LIN {X 0,Y 397.144,Z 458.266,A -85,B 0,C 180,E1 -11410.353,E2 -11410.353} C_VEL
LIN {X 0,Y 397.162,Z 458.265,A -85,B 0,C 180,E1 -11413.553,E2 -11413.553} C_VEL
LIN {X 0,Y 397.225,Z 458.255,A -85,B 0,C 180,E1 -11416.703,E2 -11416.703} C_VEL
LIN {X 0,Y 397.225,Z 458.254,A -85,B 0,C 180,E1 -11419.809,E2 -11419.809} C_VEL
LIN {X 0,Y 397.361,Z 458.247,A -85,B 0,C 180,E1 -11422.888,E2 -11422.888} C_VEL
LIN {X 0,Y 397.221,Z 458.489,A -85,B 0,C 180,E1 -11425.433,E2 -11425.433} C_VEL
LIN {X 0,Y 397.512,Z 458.679,A -85,B 0,C 180,E1 -11427.974,E2 -11427.974} C_VEL
LIN {X 0,Y 397.666,Z 458.707,A -85,B 0,C 180,E1 -11430,E2 -11430} C_VEL
LIN {X 0,Y 397.415,Z 458.63,A -85,B 0,C 180,E1 -11433.041,E2 -11433.041} C_VEL
LIN {X 0,Y 397.361,Z 458.247,A -85,B 0,C 180,E1 -11437.112,E2 -11437.112} C_VEL
LIN {X 0,Y 397.225,Z 458.255,A -85,B 0,C 180,E1 -11440.191,E2 -11440.191} C_VEL
LIN {X 0,Y 397.223,Z 458.255,A -85,B 0,C 180,E1 -11443.321,E2 -11443.321} C_VEL
LIN {X 0,Y 397.178,Z 458.26,A -85,B 0,C 180,E1 -11447.155,E2 -11447.155} C_VEL
LIN {X 0,Y 397.098,Z 458.273,A -85,B 0,C 180,E1 -11450.73,E2 -11450.73} C_VEL
LIN {X 0,Y 397.128,Z 458.267,A -85,B 0,C 180,E1 -11454.018,E2 -11454.018} C_VEL
LIN {X 0,Y 397.129,Z 458.268,A -85,B 0,C 180,E1 -11456.332,E2 -11456.332} C_VEL
LIN {X 0,Y 396.46,Z 458.351,A -85,B 0,C 180,E1 -11457.179,E2 -11457.179} C_VEL
LIN {X 0,Y 393.585,Z 458.709,A -85,B 0,C 180,E1 -11458.555,E2 -11458.555} C_VEL
LIN {X 0,Y 391.146,Z 459.012,A -85,B 0,C 180,E1 -11459.666,E2 -11459.666} C_VEL
LIN {X 0,Y 390.094,Z 459.146,A -85,B 0,C 180,E1 -11460.526,E2 -11460.526} C_VEL
LIN {X 0,Y 390.006,Z 459.152,A -85,B 0,C 180,E1 -11460.817,E2 -11460.817} C_VEL
LIN {X 0,Y 390.062,Z 459.147,A -85,B 0,C 180,E1 -11464.024,E2 -11464.024} C_VEL
LIN {X 0,Y 390.041,Z 459.151,A -85,B 0,C 180,E1 -11467.551,E2 -11467.551} C_VEL
LIN {X 0,Y 390.07,Z 459.148,A -85,B 0,C 180,E1 -11470.825,E2 -11470.825} C_VEL
LIN {X 0,Y 390.053,Z 459.149,A -85,B 0,C 180,E1 -11473.887,E2 -11473.887} C_VEL
LIN {X 0,Y 390.111,Z 459.144,A -85,B 0,C 180,E1 -11476.798,E2 -11476.798} C_VEL
LIN {X 0,Y 390.071,Z 459.147,A -85,B 0,C 180,E1 -11479.563,E2 -11479.563} C_VEL
LIN {X 0,Y 390.053,Z 459.15,A -85,B 0,C 180,E1 -11482.446,E2 -11482.446} C_VEL
LIN {X 0,Y 390.06,Z 459.104,A -85,B 0,C 180,E1 -11486.045,E2 -11486.045} C_VEL
LIN {X 0,Y 390.044,Z 459.148,A -85,B 0,C 180,E1 -11489.867,E2 -11489.867} C_VEL
LIN {X 0,Y 390.105,Z 459.094,A -85,B 0,C 180,E1 -11493.232,E2 -11493.232} C_VEL
LIN {X 0,Y 390.068,Z 459.143,A -85,B 0,C 180,E1 -11496.761,E2 -11496.761} C_VEL
LIN {X 0,Y 390.095,Z 459.132,A -85,B 0,C 180,E1 -11499.983,E2 -11499.983} C_VEL
LIN {X 0,Y 390.129,Z 459.128,A -85,B 0,C 180,E1 -11503.248,E2 -11503.248} C_VEL
LIN {X 0,Y 390.186,Z 459.129,A -85,B 0,C 180,E1 -11506.562,E2 -11506.562} C_VEL
LIN {X 0,Y 390.197,Z 459.125,A -85,B 0,C 180,E1 -11510.671,E2 -11510.671} C_VEL
LIN {X 0,Y 390.32,Z 459.1,A -85,B 0,C 180,E1 -11513.798,E2 -11513.798} C_VEL
LIN {X 0,Y 390.412,Z 459.088,A -85,B 0,C 180,E1 -11517.937,E2 -11517.937} C_VEL
LIN {X 0,Y 390.541,Z 459.084,A -85,B 0,C 180,E1 -11520,E2 -11520} C_VEL
LIN {X 0,Y 390.308,Z 459.105,A -85,B 0,C 180,E1 -11523.097,E2 -11523.097} C_VEL
LIN {X 0,Y 390.327,Z 459.112,A -85,B 0,C 180,E1 -11526.202,E2 -11526.202} C_VEL
LIN {X 0,Y 390.197,Z 459.115,A -85,B 0,C 180,E1 -11529.329,E2 -11529.329} C_VEL
LIN {X 0,Y 390.163,Z 459.123,A -85,B 0,C 180,E1 -11532.483,E2 -11532.483} C_VEL
LIN {X 0,Y 390.131,Z 459.139,A -85,B 0,C 180,E1 -11535.677,E2 -11535.677} C_VEL
LIN {X 0,Y 390.097,Z 459.098,A -85,B 0,C 180,E1 -11538.923,E2 -11538.923} C_VEL
LIN {X 0,Y 390.029,Z 459.125,A -85,B 0,C 180,E1 -11542.235,E2 -11542.235} C_VEL
LIN {X 0,Y 390.112,Z 459.13,A -85,B 0,C 180,E1 -11545.744,E2 -11545.744} C_VEL
LIN {X 0,Y 390.058,Z 459.106,A -85,B 0,C 180,E1 -11549.11,E2 -11549.11} C_VEL
LIN {X 0,Y 390.049,Z 459.145,A -85,B 0,C 180,E1 -11552.721,E2 -11552.721} C_VEL
LIN {X 0,Y 390.051,Z 459.125,A -85,B 0,C 180,E1 -11555.826,E2 -11555.826} C_VEL
LIN {X 0,Y 390.069,Z 459.129,A -85,B 0,C 180,E1 -11559.22,E2 -11559.22} C_VEL
LIN {X 0,Y 390.115,Z 459.142,A -85,B 0,C 180,E1 -11562.387,E2 -11562.387} C_VEL
LIN {X 0,Y 390.057,Z 459.139,A -85,B 0,C 180,E1 -11565.358,E2 -11565.358} C_VEL
LIN {X 0,Y 390.056,Z 459.231,A -85,B 0,C 180,E1 -11567.74,E2 -11567.74} C_VEL
LIN {X 0,Y 390.768,Z 461.893,A -85,B 0,C 180,E1 -11568.518,E2 -11568.518} C_VEL
LIN {X 0,Y 393.681,Z 471.822,A -85,B 0,C 180,E1 -11571.078,E2 -11571.078} C_VEL
LIN {X 0,Y 395.714,Z 479.188,A -85,B 0,C 180,E1 -11572.82,E2 -11572.82} C_VEL
LIN {X 0,Y 403.295,Z 494.074,A -85,B 0,C 180,E1 -11573.969,E2 -11573.969} C_VEL
LIN {X 0,Y 409.389,Z 507.007,A -85,B 0,C 180,E1 -11574.853,E2 -11574.853} C_VEL
LIN {X 0,Y 414.14,Z 527.273,A -85,B 0,C 180,E1 -11575.728,E2 -11575.728} C_VEL
LIN {X 0,Y 410.722,Z 661.42,A -85,B 0,C 180,E1 -11578.145,E2 -11578.145} C_VEL
LIN {X 0,Y 409.788,Z 693.332,A -85,B 0,C 180,E1 -11578.749,E2 -11578.749} C_VEL
LIN {X 0,Y 408.893,Z 708.266,A -85,B 0,C 180,E1 -11579.158,E2 -11579.158} C_VEL
LIN {X 0,Y 407.444,Z 726.281,A -85,B 0,C 180,E1 -11579.862,E2 -11579.862} C_VEL
LIN {X 0,Y 405.925,Z 741.244,A -85,B 0,C 180,E1 -11580.648,E2 -11580.648} C_VEL
LIN {X 0,Y 404.496,Z 753.886,A -85,B 0,C 180,E1 -11581.459,E2 -11581.459} C_VEL
LIN {X 0,Y 402.955,Z 765.529,A -85,B 0,C 180,E1 -11582.331,E2 -11582.331} C_VEL
LIN {X 0,Y 401.258,Z 777.848,A -85,B 0,C 180,E1 -11583.418,E2 -11583.418} C_VEL
LIN {X 0,Y 399.674,Z 788.357,A -85,B 0,C 180,E1 -11584.481,E2 -11584.481} C_VEL
LIN {X 0,Y 398.093,Z 798.331,A -85,B 0,C 180,E1 -11585.628,E2 -11585.628} C_VEL
LIN {X 0,Y 396.444,Z 809.034,A -85,B 0,C 180,E1 -11587.046,E2 -11587.046} C_VEL
LIN {X 0,Y 394.852,Z 819.246,A -85,B 0,C 180,E1 -11588.6,E2 -11588.6} C_VEL
LIN {X 0,Y 393.427,Z 828.207,A -85,B 0,C 180,E1 -11590.16,E2 -11590.16} C_VEL
LIN {X 0,Y 392.277,Z 836.067,A -85,B 0,C 180,E1 -11591.721,E2 -11591.721} C_VEL
LIN {X 0,Y 391.408,Z 843.069,A -85,B 0,C 180,E1 -11593.305,E2 -11593.305} C_VEL
LIN {X 0,Y 390.552,Z 849.207,A -85,B 0,C 180,E1 -11594.875,E2 -11594.875} C_VEL
LIN {X 0,Y 389.788,Z 856.132,A -85,B 0,C 180,E1 -11596.968,E2 -11596.968} C_VEL
LIN {X 0,Y 389.223,Z 861.906,A -85,B 0,C 180,E1 -11599.071,E2 -11599.071} C_VEL
LIN {X 0,Y 388.948,Z 865.514,A -85,B 0,C 180,E1 -11600.641,E2 -11600.641} C_VEL
LIN {X 0,Y 388.809,Z 869.361,A -85,B 0,C 180,E1 -11602.731,E2 -11602.731} C_VEL
LIN {X 0,Y 388.736,Z 871.161,A -85,B 0,C 180,E1 -11603.905,E2 -11603.905} C_VEL
LIN {X 0,Y 388.656,Z 873.336,A -85,B 0,C 180,E1 -11605.852,E2 -11605.852} C_VEL
LIN {X 0,Y 388.649,Z 874.754,A -85,B 0,C 180,E1 -11607.927,E2 -11607.927} C_VEL
LIN {X 0,Y 388.671,Z 875.226,A -85,B 0,C 180,E1 -11610,E2 -11610} C_VEL
LIN {X 0,Y 388.649,Z 874.754,A -85,B 0,C 180,E1 -11612.073,E2 -11612.073} C_VEL
LIN {X 0,Y 388.656,Z 873.336,A -85,B 0,C 180,E1 -11614.148,E2 -11614.148} C_VEL
LIN {X 0,Y 388.757,Z 870.959,A -85,B 0,C 180,E1 -11616.227,E2 -11616.227} C_VEL
LIN {X 0,Y 388.897,Z 866.553,A -85,B 0,C 180,E1 -11618.836,E2 -11618.836} C_VEL
LIN {X 0,Y 389.063,Z 863.189,A -85,B 0,C 180,E1 -11620.407,E2 -11620.407} C_VEL
LIN {X 0,Y 389.627,Z 857.696,A -85,B 0,C 180,E1 -11622.501,E2 -11622.501} C_VEL
LIN {X 0,Y 390.134,Z 852.84,A -85,B 0,C 180,E1 -11624.075,E2 -11624.075} C_VEL
LIN {X 0,Y 391.062,Z 845.173,A -85,B 0,C 180,E1 -11626.174,E2 -11626.174} C_VEL
LIN {X 0,Y 391.964,Z 838.521,A -85,B 0,C 180,E1 -11627.746,E2 -11627.746} C_VEL
LIN {X 0,Y 393.005,Z 830.965,A -85,B 0,C 180,E1 -11629.319,E2 -11629.319} C_VEL
LIN {X 0,Y 394.321,Z 822.378,A -85,B 0,C 180,E1 -11630.883,E2 -11630.883} C_VEL
LIN {X 0,Y 395.742,Z 813.648,A -85,B 0,C 180,E1 -11632.282,E2 -11632.282} C_VEL
LIN {X 0,Y 397.465,Z 802.359,A -85,B 0,C 180,E1 -11633.858,E2 -11633.858} C_VEL
LIN {X 0,Y 398.918,Z 792.932,A -85,B 0,C 180,E1 -11635.012,E2 -11635.012} C_VEL
LIN {X 0,Y 400.659,Z 781.957,A -85,B 0,C 180,E1 -11636.184,E2 -11636.184} C_VEL
LIN {X 0,Y 402.337,Z 770.031,A -85,B 0,C 180,E1 -11637.292,E2 -11637.292} C_VEL
LIN {X 0,Y 403.98,Z 757.368,A -85,B 0,C 180,E1 -11638.298,E2 -11638.298} C_VEL
LIN {X 0,Y 405.41,Z 746.377,A -85,B 0,C 180,E1 -11639.038,E2 -11639.038} C_VEL
LIN {X 0,Y 406.742,Z 733.374,A -85,B 0,C 180,E1 -11639.785,E2 -11639.785} C_VEL
LIN {X 0,Y 408.03,Z 719.739,A -85,B 0,C 180,E1 -11640.414,E2 -11640.414} C_VEL
LIN {X 0,Y 409.047,Z 706.438,A -85,B 0,C 180,E1 -11640.895,E2 -11640.895} C_VEL
LIN {X 0,Y 409.807,Z 693.333,A -85,B 0,C 180,E1 -11641.249,E2 -11641.249} C_VEL
LIN {X 0,Y 410.809,Z 657.838,A -85,B 0,C 180,E1 -11641.919,E2 -11641.919} C_VEL
LIN {X 0,Y 414.182,Z 528.831,A -85,B 0,C 180,E1 -11644.236,E2 -11644.236} C_VEL
LIN {X 0,Y 413.765,Z 525.616,A -85,B 0,C 180,E1 -11644.341,E2 -11644.341} C_VEL
LIN {X 0,Y 409.15,Z 506.188,A -85,B 0,C 180,E1 -11645.187,E2 -11645.187} C_VEL
LIN {X 0,Y 399.516,Z 486.667,A -85,B 0,C 180,E1 -11646.585,E2 -11646.585} C_VEL
LIN {X 0,Y 395.6,Z 479.006,A -85,B 0,C 180,E1 -11647.209,E2 -11647.209} C_VEL
LIN {X 0,Y 392.819,Z 468.701,A -85,B 0,C 180,E1 -11649.707,E2 -11649.707} C_VEL
LIN {X 0,Y 390.089,Z 459.484,A -85,B 0,C 180,E1 -11652.144,E2 -11652.144} C_VEL
LIN {X 0,Y 390.037,Z 459.16,A -85,B 0,C 180,E1 -11652.373,E2 -11652.373} C_VEL
LIN {X 0,Y 390.097,Z 459.126,A -85,B 0,C 180,E1 -11656.106,E2 -11656.106} C_VEL
LIN {X 0,Y 390.077,Z 459.128,A -85,B 0,C 180,E1 -11659.174,E2 -11659.174} C_VEL
LIN {X 0,Y 390.041,Z 459.15,A -85,B 0,C 180,E1 -11662.448,E2 -11662.448} C_VEL
LIN {X 0,Y 390.062,Z 459.124,A -85,B 0,C 180,E1 -11666.045,E2 -11666.045} C_VEL
LIN {X 0,Y 390.041,Z 459.147,A -85,B 0,C 180,E1 -11668.497,E2 -11668.497} C_VEL
LIN {X 0,Y 390.111,Z 459.096,A -85,B 0,C 180,E1 -11672.069,E2 -11672.069} C_VEL
LIN {X 0,Y 390.07,Z 459.145,A -85,B 0,C 180,E1 -11675.519,E2 -11675.519} C_VEL
LIN {X 0,Y 390.047,Z 459.102,A -85,B 0,C 180,E1 -11678.877,E2 -11678.877} C_VEL
LIN {X 0,Y 390.12,Z 459.115,A -85,B 0,C 180,E1 -11682.166,E2 -11682.166} C_VEL
LIN {X 0,Y 390.136,Z 459.132,A -85,B 0,C 180,E1 -11685.392,E2 -11685.392} C_VEL
LIN {X 0,Y 390.142,Z 459.138,A -85,B 0,C 180,E1 -11688.571,E2 -11688.571} C_VEL
LIN {X 0,Y 390.3,Z 459.103,A -85,B 0,C 180,E1 -11692.031,E2 -11692.031} C_VEL
LIN {X 0,Y 390.223,Z 459.122,A -85,B 0,C 180,E1 -11694.833,E2 -11694.833} C_VEL
LIN {X 0,Y 390.412,Z 459.097,A -85,B 0,C 180,E1 -11697.937,E2 -11697.937} C_VEL
LIN {X 0,Y 390.541,Z 459.083,A -85,B 0,C 180,E1 -11700,E2 -11700} C_VEL
LIN {X 0,Y 390.308,Z 459.113,A -85,B 0,C 180,E1 -11703.096,E2 -11703.096} C_VEL
LIN {X 0,Y 390.295,Z 459.102,A -85,B 0,C 180,E1 -11706.61,E2 -11706.61} C_VEL
LIN {X 0,Y 390.197,Z 459.124,A -85,B 0,C 180,E1 -11709.329,E2 -11709.329} C_VEL
LIN {X 0,Y 390.186,Z 459.129,A -85,B 0,C 180,E1 -11713.438,E2 -11713.438} C_VEL
LIN {X 0,Y 390.14,Z 459.137,A -85,B 0,C 180,E1 -11717.308,E2 -11717.308} C_VEL
LIN {X 0,Y 390.079,Z 459.133,A -85,B 0,C 180,E1 -11720.47,E2 -11720.47} C_VEL
LIN {X 0,Y 390.065,Z 459.142,A -85,B 0,C 180,E1 -11723.352,E2 -11723.352} C_VEL
LIN {X 0,Y 390.105,Z 459.094,A -85,B 0,C 180,E1 -11726.768,E2 -11726.768} C_VEL
LIN {X 0,Y 390.036,Z 459.15,A -85,B 0,C 180,E1 -11730.299,E2 -11730.299} C_VEL
LIN {X 0,Y 390.06,Z 459.104,A -85,B 0,C 180,E1 -11734.025,E2 -11734.025} C_VEL
LIN {X 0,Y 390.053,Z 459.15,A -85,B 0,C 180,E1 -11737.554,E2 -11737.554} C_VEL
LIN {X 0,Y 390.076,Z 459.147,A -85,B 0,C 180,E1 -11740.826,E2 -11740.826} C_VEL
LIN {X 0,Y 390.099,Z 459.143,A -85,B 0,C 180,E1 -11743.894,E2 -11743.894} C_VEL
LIN {X 0,Y 390.074,Z 459.148,A -85,B 0,C 180,E1 -11747.62,E2 -11747.62} C_VEL
LIN {X 0,Y 390.089,Z 459.146,A -85,B 0,C 180,E1 -11750.909,E2 -11750.909} C_VEL
LIN {X 0,Y 390.08,Z 459.145,A -85,B 0,C 180,E1 -11754.794,E2 -11754.794} C_VEL
LIN {X 0,Y 390.018,Z 459.152,A -85,B 0,C 180,E1 -11758.496,E2 -11758.496} C_VEL
LIN {X 0,Y 390.112,Z 459.143,A -85,B 0,C 180,E1 -11762.07,E2 -11762.07} C_VEL
LIN {X 0,Y 390.076,Z 459.145,A -85,B 0,C 180,E1 -11765.52,E2 -11765.52} C_VEL
LIN {X 0,Y 390.051,Z 459.149,A -85,B 0,C 180,E1 -11768.878,E2 -11768.878} C_VEL
LIN {X 0,Y 390.124,Z 459.142,A -85,B 0,C 180,E1 -11772.167,E2 -11772.167} C_VEL
LIN {X 0,Y 390.173,Z 459.305,A -85,B 0,C 180,E1 -11775.527,E2 -11775.527} C_VEL
LIN {X 0,Y 390.554,Z 460.669,A -85,B 0,C 180,E1 -11776.957,E2 -11776.957} C_VEL
LIN {X 0,Y 391.562,Z 462.574,A -85,B 0,C 180,E1 -11778.351,E2 -11778.351} C_VEL
LIN {X 0,Y 392.987,Z 463.95,A -85,B 0,C 180,E1 -11780.31,E2 -11780.31} C_VEL
LIN {X 0,Y 394.469,Z 464.73,A -85,B 0,C 180,E1 -11782.836,E2 -11782.836} C_VEL
LIN {X 0,Y 395.521,Z 465.381,A -85,B 0,C 180,E1 -11785.414,E2 -11785.414} C_VEL
LIN {X 0,Y 396.123,Z 465.642,A -85,B 0,C 180,E1 -11787.967,E2 -11787.967} C_VEL
LIN {X 0,Y 396.315,Z 465.672,A -85,B 0,C 180,E1 -11790,E2 -11790} C_VEL
LIN {X 0,Y 396.123,Z 465.642,A -85,B 0,C 180,E1 -11792.033,E2 -11792.033} C_VEL
LIN {X 0,Y 395.52,Z 465.38,A -85,B 0,C 180,E1 -11794.586,E2 -11794.586} C_VEL
LIN {X 0,Y 394.468,Z 464.729,A -85,B 0,C 180,E1 -11797.164,E2 -11797.164} C_VEL
LIN {X 0,Y 392.881,Z 463.843,A -85,B 0,C 180,E1 -11799.836,E2 -11799.836} C_VEL
LIN {X 0,Y 391.466,Z 462.435,A -85,B 0,C 180,E1 -11801.783,E2 -11801.783} C_VEL
LIN {X 0,Y 390.268,Z 459.788,A -85,B 0,C 180,E1 -11803.804,E2 -11803.804} C_VEL
LIN {X 0,Y 390.125,Z 459.18,A -85,B 0,C 180,E1 -11805.142,E2 -11805.142} C_VEL
LIN {X 0,Y 390.124,Z 459.141,A -85,B 0,C 180,E1 -11807.833,E2 -11807.833} C_VEL
LIN {X 0,Y 390.051,Z 459.149,A -85,B 0,C 180,E1 -11811.122,E2 -11811.122} C_VEL
LIN {X 0,Y 390.075,Z 459.146,A -85,B 0,C 180,E1 -11814.48,E2 -11814.48} C_VEL
LIN {X 0,Y 390.112,Z 459.143,A -85,B 0,C 180,E1 -11817.93,E2 -11817.93} C_VEL
LIN {X 0,Y 390.006,Z 459.152,A -85,B 0,C 180,E1 -11820.817,E2 -11820.817} C_VEL
LIN {X 0,Y 389.333,Z 459.239,A -85,B 0,C 180,E1 -11821.679,E2 -11821.679} C_VEL
LIN {X 0,Y 386.485,Z 459.594,A -85,B 0,C 180,E1 -11823.081,E2 -11823.081} C_VEL
LIN {X 0,Y 384.087,Z 459.891,A -85,B 0,C 180,E1 -11824.214,E2 -11824.214} C_VEL
LIN {X 0,Y 383.07,Z 460.019,A -85,B 0,C 180,E1 -11825.09,E2 -11825.09} C_VEL
LIN {X 0,Y 382.993,Z 460.025,A -85,B 0,C 180,E1 -11825.386,E2 -11825.386} C_VEL
LIN {X 0,Y 383.002,Z 460.027,A -85,B 0,C 180,E1 -11828.6,E2 -11828.6} C_VEL
LIN {X 0,Y 383.007,Z 460.025,A -85,B 0,C 180,E1 -11831.343,E2 -11831.343} C_VEL
LIN {X 0,Y 383.001,Z 460.027,A -85,B 0,C 180,E1 -11834.305,E2 -11834.305} C_VEL
LIN {X 0,Y 383.068,Z 460.02,A -85,B 0,C 180,E1 -11837.249,E2 -11837.249} C_VEL
LIN {X 0,Y 383.015,Z 460.026,A -85,B 0,C 180,E1 -11840.412,E2 -11840.412} C_VEL
LIN {X 0,Y 383.019,Z 460.006,A -85,B 0,C 180,E1 -11844.044,E2 -11844.044} C_VEL
LIN {X 0,Y 382.98,Z 460.004,A -85,B 0,C 180,E1 -11847.577,E2 -11847.577} C_VEL
LIN {X 0,Y 382.99,Z 460.027,A -85,B 0,C 180,E1 -11850.3,E2 -11850.3} C_VEL
LIN {X 0,Y 383.049,Z 459.974,A -85,B 0,C 180,E1 -11852.698,E2 -11852.698} C_VEL
LIN {X 0,Y 383.042,Z 459.992,A -85,B 0,C 180,E1 -11855.039,E2 -11855.039} C_VEL
LIN {X 0,Y 382.984,Z 460.026,A -85,B 0,C 180,E1 -11858.469,E2 -11858.469} C_VEL
LIN {X 0,Y 383.081,Z 460.016,A -85,B 0,C 180,E1 -11861.828,E2 -11861.828} C_VEL
LIN {X 0,Y 383.101,Z 460.003,A -85,B 0,C 180,E1 -11865.118,E2 -11865.118} C_VEL
LIN {X 0,Y 383.089,Z 460.001,A -85,B 0,C 180,E1 -11868.358,E2 -11868.358} C_VEL
LIN {X 0,Y 383.256,Z 459.988,A -85,B 0,C 180,E1 -11871.975,E2 -11871.975} C_VEL
LIN {X 0,Y 383.193,Z 459.993,A -85,B 0,C 180,E1 -11874.739,E2 -11874.739} C_VEL
LIN {X 0,Y 383.38,Z 459.964,A -85,B 0,C 180,E1 -11877.899,E2 -11877.899} C_VEL
LIN {X 0,Y 383.511,Z 459.96,A -85,B 0,C 180,E1 -11880,E2 -11880} C_VEL
LIN {X 0,Y 383.244,Z 459.984,A -85,B 0,C 180,E1 -11883.154,E2 -11883.154} C_VEL
LIN {X 0,Y 383.281,Z 459.989,A -85,B 0,C 180,E1 -11886.317,E2 -11886.317} C_VEL
LIN {X 0,Y 383.144,Z 459.996,A -85,B 0,C 180,E1 -11889.502,E2 -11889.502} C_VEL
LIN {X 0,Y 383.118,Z 459.997,A -85,B 0,C 180,E1 -11893.536,E2 -11893.536} C_VEL
LIN {X 0,Y 383.087,Z 459.997,A -85,B 0,C 180,E1 -11897.455,E2 -11897.455} C_VEL
LIN {X 0,Y 383.021,Z 459.97,A -85,B 0,C 180,E1 -11900.647,E2 -11900.647} C_VEL
LIN {X 0,Y 383.018,Z 460.023,A -85,B 0,C 180,E1 -11903.808,E2 -11903.808} C_VEL
LIN {X 0,Y 383.073,Z 460,A -85,B 0,C 180,E1 -11906.124,E2 -11906.124} C_VEL
LIN {X 0,Y 383.043,Z 459.974,A -85,B 0,C 180,E1 -11908.493,E2 -11908.493} C_VEL
LIN {X 0,Y 383.002,Z 460.025,A -85,B 0,C 180,E1 -11912.428,E2 -11912.428} C_VEL
LIN {X 0,Y 383.021,Z 460.001,A -85,B 0,C 180,E1 -11915.956,E2 -11915.956} C_VEL
LIN {X 0,Y 383.017,Z 460.003,A -85,B 0,C 180,E1 -11919.588,E2 -11919.588} C_VEL
LIN {X 0,Y 383.061,Z 460.016,A -85,B 0,C 180,E1 -11922.789,E2 -11922.789} C_VEL
LIN {X 0,Y 383.01,Z 460.02,A -85,B 0,C 180,E1 -11926.522,E2 -11926.522} C_VEL
LIN {X 0,Y 383.036,Z 460.276,A -85,B 0,C 180,E1 -11927.147,E2 -11927.147} C_VEL
LIN {X 0,Y 386.351,Z 471.502,A -85,B 0,C 180,E1 -11930.189,E2 -11930.189} C_VEL
LIN {X 0,Y 388.322,Z 478.732,A -85,B 0,C 180,E1 -11931.974,E2 -11931.974} C_VEL
LIN {X 0,Y 397.62,Z 496.664,A -85,B 0,C 180,E1 -11933.433,E2 -11933.433} C_VEL
LIN {X 0,Y 403.932,Z 510.042,A -85,B 0,C 180,E1 -11934.376,E2 -11934.376} C_VEL
LIN {X 0,Y 408.265,Z 528.969,A -85,B 0,C 180,E1 -11935.204,E2 -11935.204} C_VEL
LIN {X 0,Y 404.323,Z 675.539,A -85,B 0,C 180,E1 -11937.875,E2 -11937.875} C_VEL
LIN {X 0,Y 403.49,Z 698.576,A -85,B 0,C 180,E1 -11938.352,E2 -11938.352} C_VEL
LIN {X 0,Y 402.19,Z 715.47,A -85,B 0,C 180,E1 -11938.903,E2 -11938.903} C_VEL
LIN {X 0,Y 401.069,Z 728.224,A -85,B 0,C 180,E1 -11939.459,E2 -11939.459} C_VEL
LIN {X 0,Y 399.722,Z 741.033,A -85,B 0,C 180,E1 -11940.146,E2 -11940.146} C_VEL
LIN {X 0,Y 398.23,Z 753.675,A -85,B 0,C 180,E1 -11940.967,E2 -11940.967} C_VEL
LIN {X 0,Y 396.63,Z 765.317,A -85,B 0,C 180,E1 -11941.851,E2 -11941.851} C_VEL
LIN {X 0,Y 394.824,Z 777.635,A -85,B 0,C 180,E1 -11942.95,E2 -11942.95} C_VEL
LIN {X 0,Y 393.218,Z 788.145,A -85,B 0,C 180,E1 -11944.031,E2 -11944.031} C_VEL
LIN {X 0,Y 391.37,Z 799.125,A -85,B 0,C 180,E1 -11945.323,E2 -11945.323} C_VEL
LIN {X 0,Y 389.803,Z 808.82,A -85,B 0,C 180,E1 -11946.632,E2 -11946.632} C_VEL
LIN {X 0,Y 388.132,Z 819.033,A -85,B 0,C 180,E1 -11948.211,E2 -11948.211} C_VEL
LIN {X 0,Y 386.63,Z 827.993,A -85,B 0,C 180,E1 -11949.796,E2 -11949.796} C_VEL
LIN {X 0,Y 385.34,Z 836.439,A -85,B 0,C 180,E1 -11951.513,E2 -11951.513} C_VEL
LIN {X 0,Y 384.323,Z 843.908,A -85,B 0,C 180,E1 -11953.261,E2 -11953.261} C_VEL
LIN {X 0,Y 383.353,Z 850.811,A -85,B 0,C 180,E1 -11955.128,E2 -11955.128} C_VEL
LIN {X 0,Y 382.823,Z 855.709,A -85,B 0,C 180,E1 -11956.653,E2 -11956.653} C_VEL
LIN {X 0,Y 382.318,Z 860.408,A -85,B 0,C 180,E1 -11958.334,E2 -11958.334} C_VEL
LIN {X 0,Y 381.887,Z 865.303,A -85,B 0,C 180,E1 -11960.466,E2 -11960.466} C_VEL
LIN {X 0,Y 381.711,Z 869.149,A -85,B 0,C 180,E1 -11962.595,E2 -11962.595} C_VEL
LIN {X 0,Y 381.655,Z 871.134,A -85,B 0,C 180,E1 -11963.924,E2 -11963.924} C_VEL
LIN {X 0,Y 381.581,Z 873.126,A -85,B 0,C 180,E1 -11965.775,E2 -11965.775} C_VEL
LIN {X 0,Y 381.547,Z 874.544,A -85,B 0,C 180,E1 -11967.889,E2 -11967.889} C_VEL
LIN {X 0,Y 381.586,Z 875.016,A -85,B 0,C 180,E1 -11970,E2 -11970} C_VEL
LIN {X 0,Y 381.547,Z 874.544,A -85,B 0,C 180,E1 -11972.111,E2 -11972.111} C_VEL
LIN {X 0,Y 381.581,Z 873.126,A -85,B 0,C 180,E1 -11974.225,E2 -11974.225} C_VEL
LIN {X 0,Y 381.662,Z 870.748,A -85,B 0,C 180,E1 -11976.343,E2 -11976.343} C_VEL
LIN {X 0,Y 381.819,Z 866.341,A -85,B 0,C 180,E1 -11979.001,E2 -11979.001} C_VEL
LIN {X 0,Y 382.021,Z 862.977,A -85,B 0,C 180,E1 -11980.601,E2 -11980.601} C_VEL
LIN {X 0,Y 382.59,Z 857.483,A -85,B 0,C 180,E1 -11982.734,E2 -11982.734} C_VEL
LIN {X 0,Y 383.157,Z 852.627,A -85,B 0,C 180,E1 -11984.336,E2 -11984.336} C_VEL
LIN {X 0,Y 384.151,Z 844.96,A -85,B 0,C 180,E1 -11986.473,E2 -11986.473} C_VEL
LIN {X 0,Y 385.082,Z 838.307,A -85,B 0,C 180,E1 -11988.075,E2 -11988.075} C_VEL
LIN {X 0,Y 386.184,Z 830.751,A -85,B 0,C 180,E1 -11989.674,E2 -11989.674} C_VEL
LIN {X 0,Y 387.58,Z 822.165,A -85,B 0,C 180,E1 -11991.263,E2 -11991.263} C_VEL
LIN {X 0,Y 389.242,Z 812.49,A -85,B 0,C 180,E1 -11992.823,E2 -11992.823} C_VEL
LIN {X 0,Y 390.871,Z 802.146,A -85,B 0,C 180,E1 -11994.286,E2 -11994.286} C_VEL
LIN {X 0,Y 392.409,Z 792.72,A -85,B 0,C 180,E1 -11995.457,E2 -11995.457} C_VEL
LIN {X 0,Y 394.393,Z 780.55,A -85,B 0,C 180,E1 -11996.763,E2 -11996.763} C_VEL
LIN {X 0,Y 396.139,Z 768.316,A -85,B 0,C 180,E1 -11997.899,E2 -11997.899} C_VEL
LIN {X 0,Y 397.693,Z 757.156,A -85,B 0,C 180,E1 -11998.787,E2 -11998.787} C_VEL
LIN {X 0,Y 399.277,Z 745.139,A -85,B 0,C 180,E1 -11999.6,E2 -11999.6} C_VEL
LIN {X 0,Y 400.569,Z 733.163,A -85,B 0,C 180,E1 -12000.292,E2 -12000.292} C_VEL
LIN {X 0,Y 401.864,Z 719.795,A -85,B 0,C 180,E1 -12000.919,E2 -12000.919} C_VEL
LIN {X 0,Y 402.944,Z 706.567,A -85,B 0,C 180,E1 -12001.403,E2 -12001.403} C_VEL
LIN {X 0,Y 403.749,Z 693.123,A -85,B 0,C 180,E1 -12001.772,E2 -12001.772} C_VEL
LIN {X 0,Y 404.797,Z 657.628,A -85,B 0,C 180,E1 -12002.451,E2 -12002.451} C_VEL
LIN {X 0,Y 408.007,Z 538.652,A -85,B 0,C 180,E1 -12004.618,E2 -12004.618} C_VEL
LIN {X 0,Y 408.138,Z 528.273,A -85,B 0,C 180,E1 -12004.823,E2 -12004.823} C_VEL
LIN {X 0,Y 403.786,Z 509.589,A -85,B 0,C 180,E1 -12005.649,E2 -12005.649} C_VEL
LIN {X 0,Y 394.84,Z 491.255,A -85,B 0,C 180,E1 -12006.985,E2 -12006.985} C_VEL
LIN {X 0,Y 388.337,Z 478.732,A -85,B 0,C 180,E1 -12008.024,E2 -12008.024} C_VEL
LIN {X 0,Y 385.267,Z 467.825,A -85,B 0,C 180,E1 -12010.778,E2 -12010.778} C_VEL
LIN {X 0,Y 383.061,Z 460.454,A -85,B 0,C 180,E1 -12012.788,E2 -12012.788} C_VEL
LIN {X 0,Y 383.027,Z 460.016,A -85,B 0,C 180,E1 -12013.114,E2 -12013.114} C_VEL
LIN {X 0,Y 383.033,Z 460.004,A -85,B 0,C 180,E1 -12015.794,E2 -12015.794} C_VEL
LIN {X 0,Y 383.039,Z 460.009,A -85,B 0,C 180,E1 -12018.786,E2 -12018.786} C_VEL
LIN {X 0,Y 382.998,Z 460.028,A -85,B 0,C 180,E1 -12022.095,E2 -12022.095} C_VEL
LIN {X 0,Y 383.012,Z 459.995,A -85,B 0,C 180,E1 -12025.331,E2 -12025.331} C_VEL
LIN {X 0,Y 383.03,Z 460.025,A -85,B 0,C 180,E1 -12027.852,E2 -12027.852} C_VEL
LIN {X 0,Y 383.057,Z 459.972,A -85,B 0,C 180,E1 -12031.72,E2 -12031.72} C_VEL
LIN {X 0,Y 383.044,Z 460.019,A -85,B 0,C 180,E1 -12035.039,E2 -12035.039} C_VEL
LIN {X 0,Y 382.984,Z 459.987,A -85,B 0,C 180,E1 -12038.468,E2 -12038.468} C_VEL
LIN {X 0,Y 383.081,Z 459.986,A -85,B 0,C 180,E1 -12041.827,E2 -12041.827} C_VEL
LIN {X 0,Y 383.102,Z 460.008,A -85,B 0,C 180,E1 -12045.118,E2 -12045.118} C_VEL
LIN {X 0,Y 383.091,Z 460.012,A -85,B 0,C 180,E1 -12048.358,E2 -12048.358} C_VEL
LIN {X 0,Y 383.256,Z 459.979,A -85,B 0,C 180,E1 -12051.975,E2 -12051.975} C_VEL
LIN {X 0,Y 383.195,Z 459.998,A -85,B 0,C 180,E1 -12054.738,E2 -12054.738} C_VEL
LIN {X 0,Y 383.379,Z 459.973,A -85,B 0,C 180,E1 -12057.899,E2 -12057.899} C_VEL
LIN {X 0,Y 383.511,Z 459.958,A -85,B 0,C 180,E1 -12060,E2 -12060} C_VEL
LIN {X 0,Y 383.245,Z 459.992,A -85,B 0,C 180,E1 -12063.153,E2 -12063.153} C_VEL
LIN {X 0,Y 383.255,Z 459.978,A -85,B 0,C 180,E1 -12066.602,E2 -12066.602} C_VEL
LIN {X 0,Y 383.143,Z 460.002,A -85,B 0,C 180,E1 -12069.502,E2 -12069.502} C_VEL
LIN {X 0,Y 383.117,Z 460.009,A -85,B 0,C 180,E1 -12073.536,E2 -12073.536} C_VEL
LIN {X 0,Y 383.086,Z 460.015,A -85,B 0,C 180,E1 -12077.454,E2 -12077.454} C_VEL
LIN {X 0,Y 383.02,Z 460.012,A -85,B 0,C 180,E1 -12080.647,E2 -12080.647} C_VEL
LIN {X 0,Y 383.017,Z 460.018,A -85,B 0,C 180,E1 -12083.808,E2 -12083.808} C_VEL
LIN {X 0,Y 383.072,Z 459.97,A -85,B 0,C 180,E1 -12086.123,E2 -12086.123} C_VEL
LIN {X 0,Y 383.042,Z 459.996,A -85,B 0,C 180,E1 -12088.492,E2 -12088.492} C_VEL
LIN {X 0,Y 383.003,Z 460.008,A -85,B 0,C 180,E1 -12092.15,E2 -12092.15} C_VEL
LIN {X 0,Y 383.01,Z 459.984,A -85,B 0,C 180,E1 -12094.668,E2 -12094.668} C_VEL
LIN {X 0,Y 383.003,Z 460.027,A -85,B 0,C 180,E1 -12097.906,E2 -12097.906} C_VEL
LIN {X 0,Y 383.04,Z 460.024,A -85,B 0,C 180,E1 -12101.339,E2 -12101.339} C_VEL
LIN {X 0,Y 383.03,Z 460.023,A -85,B 0,C 180,E1 -12104.31,E2 -12104.31} C_VEL
LIN {X 0,Y 383.033,Z 460.023,A -85,B 0,C 180,E1 -12107.245,E2 -12107.245} C_VEL
LIN {X 0,Y 383.015,Z 460.025,A -85,B 0,C 180,E1 -12110.413,E2 -12110.413} C_VEL
LIN {X 0,Y 383.021,Z 460.024,A -85,B 0,C 180,E1 -12114.045,E2 -12114.045} C_VEL
LIN {X 0,Y 382.981,Z 460.03,A -85,B 0,C 180,E1 -12117.578,E2 -12117.578} C_VEL
LIN {X 0,Y 382.987,Z 460.028,A -85,B 0,C 180,E1 -12120.3,E2 -12120.3} C_VEL
LIN {X 0,Y 383.076,Z 460.017,A -85,B 0,C 180,E1 -12124.021,E2 -12124.021} C_VEL
LIN {X 0,Y 383.004,Z 460.026,A -85,B 0,C 180,E1 -12127.336,E2 -12127.336} C_VEL
LIN {X 0,Y 383.089,Z 460.2,A -85,B 0,C 180,E1 -12130.021,E2 -12130.021} C_VEL
LIN {X 0,Y 383.447,Z 461.553,A -85,B 0,C 180,E1 -12131.015,E2 -12131.015} C_VEL
LIN {X 0,Y 384.784,Z 463.815,A -85,B 0,C 180,E1 -12132.232,E2 -12132.232} C_VEL
LIN {X 0,Y 386.964,Z 465.493,A -85,B 0,C 180,E1 -12134.192,E2 -12134.192} C_VEL
LIN {X 0,Y 388.846,Z 466.639,A -85,B 0,C 180,E1 -12136.011,E2 -12136.011} C_VEL
LIN {X 0,Y 390.564,Z 469.516,A -85,B 0,C 180,E1 -12138.189,E2 -12138.189} C_VEL
LIN {X 0,Y 392.123,Z 470.995,A -85,B 0,C 180,E1 -12140.317,E2 -12140.317} C_VEL
LIN {X 0,Y 393.591,Z 471.775,A -85,B 0,C 180,E1 -12142.82,E2 -12142.82} C_VEL
LIN {X 0,Y 394.492,Z 472.245,A -85,B 0,C 180,E1 -12144.89,E2 -12144.89} C_VEL
LIN {X 0,Y 394.837,Z 472.584,A -85,B 0,C 180,E1 -12145.917,E2 -12145.917} C_VEL
LIN {X 0,Y 395.257,Z 472.689,A -85,B 0,C 180,E1 -12147.962,E2 -12147.962} C_VEL
LIN {X 0,Y 395.45,Z 472.72,A -85,B 0,C 180,E1 -12150,E2 -12150} C_VEL
LIN {X 0,Y 395.258,Z 472.69,A -85,B 0,C 180,E1 -12152.038,E2 -12152.038} C_VEL
LIN {X 0,Y 394.65,Z 472.428,A -85,B 0,C 180,E1 -12154.596,E2 -12154.596} C_VEL
LIN {X 0,Y 393.591,Z 471.772,A -85,B 0,C 180,E1 -12157.18,E2 -12157.18} C_VEL
LIN {X 0,Y 391.99,Z 470.903,A -85,B 0,C 180,E1 -12159.859,E2 -12159.859} C_VEL
LIN {X 0,Y 390.47,Z 469.378,A -85,B 0,C 180,E1 -12161.946,E2 -12161.946} C_VEL
LIN {X 0,Y 388.845,Z 466.637,A -85,B 0,C 180,E1 -12163.989,E2 -12163.989} C_VEL
LIN {X 0,Y 386.032,Z 464.937,A -85,B 0,C 180,E1 -12166.662,E2 -12166.662} C_VEL
LIN {X 0,Y 384.202,Z 463.095,A -85,B 0,C 180,E1 -12168.255,E2 -12168.255} C_VEL
LIN {X 0,Y 383.196,Z 460.804,A -85,B 0,C 180,E1 -12169.415,E2 -12169.415} C_VEL
LIN {X 0,Y 383.051,Z 460.065,A -85,B 0,C 180,E1 -12170.401,E2 -12170.401} C_VEL
LIN {X 0,Y 383.029,Z 460.024,A -85,B 0,C 180,E1 -12173.807,E2 -12173.807} C_VEL
LIN {X 0,Y 383.075,Z 460.019,A -85,B 0,C 180,E1 -12176.123,E2 -12176.123} C_VEL
LIN {X 0,Y 382.987,Z 460.028,A -85,B 0,C 180,E1 -12179.7,E2 -12179.7} C_VEL
LIN {X 0,Y 382.998,Z 460.029,A -85,B 0,C 180,E1 -12183.4,E2 -12183.4} C_VEL
LIN {X 0,Y 382.993,Z 460.025,A -85,B 0,C 180,E1 -12185.386,E2 -12185.386} C_VEL
LIN {X 0,Y 382.353,Z 460.109,A -85,B 0,C 180,E1 -12186.264,E2 -12186.264} C_VEL
LIN {X 0,Y 379.545,Z 460.459,A -85,B 0,C 180,E1 -12187.692,E2 -12187.692} C_VEL
LIN {X 0,Y 377.14,Z 460.758,A -85,B 0,C 180,E1 -12188.846,E2 -12188.846} C_VEL
LIN {X 0,Y 376.085,Z 460.888,A -85,B 0,C 180,E1 -12189.738,E2 -12189.738} C_VEL
LIN {X 0,Y 375.987,Z 460.9,A -85,B 0,C 180,E1 -12190.041,E2 -12190.041} C_VEL
LIN {X 0,Y 375.939,Z 460.908,A -85,B 0,C 180,E1 -12193.763,E2 -12193.763} C_VEL
LIN {X 0,Y 375.983,Z 460.903,A -85,B 0,C 180,E1 -12196.801,E2 -12196.801} C_VEL
LIN {X 0,Y 375.992,Z 460.901,A -85,B 0,C 180,E1 -12200.027,E2 -12200.027} C_VEL
LIN {X 0,Y 375.96,Z 460.899,A -85,B 0,C 180,E1 -12203.495,E2 -12203.495} C_VEL
LIN {X 0,Y 375.952,Z 460.859,A -85,B 0,C 180,E1 -12205.888,E2 -12205.888} C_VEL
LIN {X 0,Y 375.961,Z 460.903,A -85,B 0,C 180,E1 -12209.688,E2 -12209.688} C_VEL
LIN {X 0,Y 375.994,Z 460.858,A -85,B 0,C 180,E1 -12212.142,E2 -12212.142} C_VEL
LIN {X 0,Y 375.997,Z 460.858,A -85,B 0,C 180,E1 -12214.539,E2 -12214.539} C_VEL
LIN {X 0,Y 375.95,Z 460.903,A -85,B 0,C 180,E1 -12218.045,E2 -12218.045} C_VEL
LIN {X 0,Y 376.015,Z 460.899,A -85,B 0,C 180,E1 -12221.474,E2 -12221.474} C_VEL
LIN {X 0,Y 376.05,Z 460.878,A -85,B 0,C 180,E1 -12224.833,E2 -12224.833} C_VEL
LIN {X 0,Y 376.041,Z 460.88,A -85,B 0,C 180,E1 -12228.137,E2 -12228.137} C_VEL
LIN {X 0,Y 376.211,Z 460.866,A -85,B 0,C 180,E1 -12231.918,E2 -12231.918} C_VEL
LIN {X 0,Y 376.165,Z 460.868,A -85,B 0,C 180,E1 -12234.64,E2 -12234.64} C_VEL
LIN {X 0,Y 376.346,Z 460.84,A -85,B 0,C 180,E1 -12237.86,E2 -12237.86} C_VEL
LIN {X 0,Y 376.48,Z 460.835,A -85,B 0,C 180,E1 -12240,E2 -12240} C_VEL
LIN {X 0,Y 376.182,Z 460.862,A -85,B 0,C 180,E1 -12243.213,E2 -12243.213} C_VEL
LIN {X 0,Y 376.238,Z 460.866,A -85,B 0,C 180,E1 -12246.435,E2 -12246.435} C_VEL
LIN {X 0,Y 376.111,Z 460.873,A -85,B 0,C 180,E1 -12249.682,E2 -12249.682} C_VEL
LIN {X 0,Y 376.082,Z 460.873,A -85,B 0,C 180,E1 -12253.658,E2 -12253.658} C_VEL
LIN {X 0,Y 376.036,Z 460.871,A -85,B 0,C 180,E1 -12257.608,E2 -12257.608} C_VEL
LIN {X 0,Y 375.971,Z 460.848,A -85,B 0,C 180,E1 -12260.833,E2 -12260.833} C_VEL
LIN {X 0,Y 375.983,Z 460.902,A -85,B 0,C 180,E1 -12264.282,E2 -12264.282} C_VEL
LIN {X 0,Y 376.013,Z 460.868,A -85,B 0,C 180,E1 -12266.653,E2 -12266.653} C_VEL
LIN {X 0,Y 375.97,Z 460.857,A -85,B 0,C 180,E1 -12269.079,E2 -12269.079} C_VEL
LIN {X 0,Y 375.95,Z 460.901,A -85,B 0,C 180,E1 -12272.828,E2 -12272.828} C_VEL
LIN {X 0,Y 375.952,Z 460.875,A -85,B 0,C 180,E1 -12275.416,E2 -12275.416} C_VEL
LIN {X 0,Y 375.972,Z 460.898,A -85,B 0,C 180,E1 -12278.272,E2 -12278.272} C_VEL
LIN {X 0,Y 375.985,Z 460.895,A -85,B 0,C 180,E1 -12281.611,E2 -12281.611} C_VEL
LIN {X 0,Y 375.964,Z 460.891,A -85,B 0,C 180,E1 -12285.263,E2 -12285.263} C_VEL
LIN {X 0,Y 375.961,Z 460.934,A -85,B 0,C 180,E1 -12286.315,E2 -12286.315} C_VEL
LIN {X 0,Y 376.642,Z 463.275,A -85,B 0,C 180,E1 -12287.07,E2 -12287.07} C_VEL
LIN {X 0,Y 379.946,Z 474.523,A -85,B 0,C 180,E1 -12290.141,E2 -12290.141} C_VEL
LIN {X 0,Y 381.034,Z 478.467,A -85,B 0,C 180,E1 -12291.116,E2 -12291.116} C_VEL
LIN {X 0,Y 390.84,Z 497.083,A -85,B 0,C 180,E1 -12292.707,E2 -12292.707} C_VEL
LIN {X 0,Y 398.54,Z 513.284,A -85,B 0,C 180,E1 -12293.893,E2 -12293.893} C_VEL
LIN {X 0,Y 402.372,Z 530.127,A -85,B 0,C 180,E1 -12294.648,E2 -12294.648} C_VEL
LIN {X 0,Y 398.716,Z 661,A -85,B 0,C 180,E1 -12297.067,E2 -12297.067} C_VEL
LIN {X 0,Y 397.711,Z 692.912,A -85,B 0,C 180,E1 -12297.687,E2 -12297.687} C_VEL
LIN {X 0,Y 396.76,Z 707.231,A -85,B 0,C 180,E1 -12298.083,E2 -12298.083} C_VEL
LIN {X 0,Y 395.286,Z 724.847,A -85,B 0,C 180,E1 -12298.772,E2 -12298.772} C_VEL
LIN {X 0,Y 393.541,Z 740.822,A -85,B 0,C 180,E1 -12299.629,E2 -12299.629} C_VEL
LIN {X 0,Y 392.003,Z 753.464,A -85,B 0,C 180,E1 -12300.461,E2 -12300.461} C_VEL
LIN {X 0,Y 390.313,Z 765.105,A -85,B 0,C 180,E1 -12301.354,E2 -12301.354} C_VEL
LIN {X 0,Y 388.462,Z 777.129,A -85,B 0,C 180,E1 -12302.436,E2 -12302.436} C_VEL
LIN {X 0,Y 386.781,Z 787.933,A -85,B 0,C 180,E1 -12303.566,E2 -12303.566} C_VEL
LIN {X 0,Y 384.857,Z 798.913,A -85,B 0,C 180,E1 -12304.877,E2 -12304.877} C_VEL
LIN {X 0,Y 382.999,Z 809.737,A -85,B 0,C 180,E1 -12306.374,E2 -12306.374} C_VEL
LIN {X 0,Y 381.464,Z 818.82,A -85,B 0,C 180,E1 -12307.81,E2 -12307.81} C_VEL
LIN {X 0,Y 379.87,Z 827.78,A -85,B 0,C 180,E1 -12309.42,E2 -12309.42} C_VEL
LIN {X 0,Y 378.586,Z 835.7,A -85,B 0,C 180,E1 -12311.049,E2 -12311.049} C_VEL
LIN {X 0,Y 377.572,Z 842.641,A -85,B 0,C 180,E1 -12312.674,E2 -12312.674} C_VEL
LIN {X 0,Y 376.644,Z 848.781,A -85,B 0,C 180,E1 -12314.303,E2 -12314.303} C_VEL
LIN {X 0,Y 375.762,Z 855.923,A -85,B 0,C 180,E1 -12316.549,E2 -12316.549} C_VEL
LIN {X 0,Y 375.138,Z 861.481,A -85,B 0,C 180,E1 -12318.656,E2 -12318.656} C_VEL
LIN {X 0,Y 374.812,Z 865.091,A -85,B 0,C 180,E1 -12320.285,E2 -12320.285} C_VEL
LIN {X 0,Y 374.628,Z 868.938,A -85,B 0,C 180,E1 -12322.454,E2 -12322.454} C_VEL
LIN {X 0,Y 374.5,Z 871.783,A -85,B 0,C 180,E1 -12324.616,E2 -12324.616} C_VEL
LIN {X 0,Y 374.486,Z 872.916,A -85,B 0,C 180,E1 -12325.695,E2 -12325.695} C_VEL
LIN {X 0,Y 374.446,Z 874.334,A -85,B 0,C 180,E1 -12327.849,E2 -12327.849} C_VEL
LIN {X 0,Y 374.489,Z 874.807,A -85,B 0,C 180,E1 -12330,E2 -12330} C_VEL
LIN {X 0,Y 374.446,Z 874.334,A -85,B 0,C 180,E1 -12332.151,E2 -12332.151} C_VEL
LIN {X 0,Y 374.486,Z 872.916,A -85,B 0,C 180,E1 -12334.305,E2 -12334.305} C_VEL
LIN {X 0,Y 374.563,Z 870.537,A -85,B 0,C 180,E1 -12336.464,E2 -12336.464} C_VEL
LIN {X 0,Y 374.759,Z 866.13,A -85,B 0,C 180,E1 -12339.172,E2 -12339.172} C_VEL
LIN {X 0,Y 374.987,Z 862.766,A -85,B 0,C 180,E1 -12340.802,E2 -12340.802} C_VEL
LIN {X 0,Y 375.581,Z 857.271,A -85,B 0,C 180,E1 -12342.976,E2 -12342.976} C_VEL
LIN {X 0,Y 376.173,Z 852.414,A -85,B 0,C 180,E1 -12344.609,E2 -12344.609} C_VEL
LIN {X 0,Y 377.243,Z 844.747,A -85,B 0,C 180,E1 -12346.784,E2 -12346.784} C_VEL
LIN {X 0,Y 378.22,Z 838.093,A -85,B 0,C 180,E1 -12348.414,E2 -12348.414} C_VEL
LIN {X 0,Y 379.38,Z 830.537,A -85,B 0,C 180,E1 -12350.042,E2 -12350.042} C_VEL
LIN {X 0,Y 380.871,Z 821.952,A -85,B 0,C 180,E1 -12351.656,E2 -12351.656} C_VEL
LIN {X 0,Y 382.45,Z 813.107,A -85,B 0,C 180,E1 -12353.118,E2 -12353.118} C_VEL
LIN {X 0,Y 384.339,Z 801.934,A -85,B 0,C 180,E1 -12354.726,E2 -12354.726} C_VEL
LIN {X 0,Y 385.953,Z 792.508,A -85,B 0,C 180,E1 -12355.914,E2 -12355.914} C_VEL
LIN {X 0,Y 387.847,Z 781.277,A -85,B 0,C 180,E1 -12357.147,E2 -12357.147} C_VEL
LIN {X 0,Y 389.611,Z 769.606,A -85,B 0,C 180,E1 -12358.262,E2 -12358.262} C_VEL
LIN {X 0,Y 391.441,Z 756.945,A -85,B 0,C 180,E1 -12359.291,E2 -12359.291} C_VEL
LIN {X 0,Y 393.04,Z 744.927,A -85,B 0,C 180,E1 -12360.118,E2 -12360.118} C_VEL
LIN {X 0,Y 394.553,Z 731.718,A -85,B 0,C 180,E1 -12360.878,E2 -12360.878} C_VEL
LIN {X 0,Y 395.855,Z 718.882,A -85,B 0,C 180,E1 -12361.475,E2 -12361.475} C_VEL
LIN {X 0,Y 396.924,Z 705.933,A -85,B 0,C 180,E1 -12361.951,E2 -12361.951} C_VEL
LIN {X 0,Y 397.711,Z 692.912,A -85,B 0,C 180,E1 -12362.313,E2 -12362.313} C_VEL
LIN {X 0,Y 398.83,Z 657.419,A -85,B 0,C 180,E1 -12362.998,E2 -12362.998} C_VEL
LIN {X 0,Y 402.426,Z 530.932,A -85,B 0,C 180,E1 -12365.329,E2 -12365.329} C_VEL
LIN {X 0,Y 400.188,Z 520.189,A -85,B 0,C 180,E1 -12365.787,E2 -12365.787} C_VEL
LIN {X 0,Y 398.183,Z 512.272,A -85,B 0,C 180,E1 -12366.166,E2 -12366.166} C_VEL
LIN {X 0,Y 387.908,Z 491.387,A -85,B 0,C 180,E1 -12367.751,E2 -12367.751} C_VEL
LIN {X 0,Y 381.026,Z 478.467,A -85,B 0,C 180,E1 -12368.884,E2 -12368.884} C_VEL
LIN {X 0,Y 378.068,Z 468.205,A -85,B 0,C 180,E1 -12371.564,E2 -12371.564} C_VEL
LIN {X 0,Y 376.014,Z 461.241,A -85,B 0,C 180,E1 -12373.531,E2 -12373.531} C_VEL
LIN {X 0,Y 375.958,Z 460.923,A -85,B 0,C 180,E1 -12373.761,E2 -12373.761} C_VEL
LIN {X 0,Y 375.983,Z 460.889,A -85,B 0,C 180,E1 -12376.801,E2 -12376.801} C_VEL
LIN {X 0,Y 375.993,Z 460.876,A -85,B 0,C 180,E1 -12380.027,E2 -12380.027} C_VEL
LIN {X 0,Y 375.96,Z 460.89,A -85,B 0,C 180,E1 -12383.495,E2 -12383.495} C_VEL
LIN {X 0,Y 375.955,Z 460.877,A -85,B 0,C 180,E1 -12385.888,E2 -12385.888} C_VEL
LIN {X 0,Y 375.963,Z 460.881,A -85,B 0,C 180,E1 -12389.687,E2 -12389.687} C_VEL
LIN {X 0,Y 375.995,Z 460.851,A -85,B 0,C 180,E1 -12392.141,E2 -12392.141} C_VEL
LIN {X 0,Y 375.999,Z 460.892,A -85,B 0,C 180,E1 -12394.538,E2 -12394.538} C_VEL
LIN {X 0,Y 375.95,Z 460.871,A -85,B 0,C 180,E1 -12398.045,E2 -12398.045} C_VEL
LIN {X 0,Y 376.016,Z 460.855,A -85,B 0,C 180,E1 -12401.473,E2 -12401.473} C_VEL
LIN {X 0,Y 376.05,Z 460.888,A -85,B 0,C 180,E1 -12404.832,E2 -12404.832} C_VEL
LIN {X 0,Y 376.043,Z 460.887,A -85,B 0,C 180,E1 -12408.136,E2 -12408.136} C_VEL
LIN {X 0,Y 376.211,Z 460.856,A -85,B 0,C 180,E1 -12411.918,E2 -12411.918} C_VEL
LIN {X 0,Y 376.167,Z 460.874,A -85,B 0,C 180,E1 -12414.64,E2 -12414.64} C_VEL
LIN {X 0,Y 376.346,Z 460.849,A -85,B 0,C 180,E1 -12417.859,E2 -12417.859} C_VEL
LIN {X 0,Y 376.48,Z 460.833,A -85,B 0,C 180,E1 -12420,E2 -12420} C_VEL
LIN {X 0,Y 376.183,Z 460.872,A -85,B 0,C 180,E1 -12423.213,E2 -12423.213} C_VEL
LIN {X 0,Y 376.221,Z 460.853,A -85,B 0,C 180,E1 -12426.59,E2 -12426.59} C_VEL
LIN {X 0,Y 376.111,Z 460.878,A -85,B 0,C 180,E1 -12429.681,E2 -12429.681} C_VEL
LIN {X 0,Y 376.081,Z 460.886,A -85,B 0,C 180,E1 -12433.657,E2 -12433.657} C_VEL
LIN {X 0,Y 376.036,Z 460.893,A -85,B 0,C 180,E1 -12437.607,E2 -12437.607} C_VEL
LIN {X 0,Y 375.97,Z 460.891,A -85,B 0,C 180,E1 -12440.832,E2 -12440.832} C_VEL
LIN {X 0,Y 375.981,Z 460.883,A -85,B 0,C 180,E1 -12444.282,E2 -12444.282} C_VEL
LIN {X 0,Y 376.012,Z 460.846,A -85,B 0,C 180,E1 -12446.652,E2 -12446.652} C_VEL
LIN {X 0,Y 375.969,Z 460.888,A -85,B 0,C 180,E1 -12449.079,E2 -12449.079} C_VEL
LIN {X 0,Y 375.942,Z 460.871,A -85,B 0,C 180,E1 -12452.829,E2 -12452.829} C_VEL
LIN {X 0,Y 375.951,Z 460.873,A -85,B 0,C 180,E1 -12455.416,E2 -12455.416} C_VEL
LIN {X 0,Y 375.975,Z 460.902,A -85,B 0,C 180,E1 -12458.272,E2 -12458.272} C_VEL
LIN {X 0,Y 375.983,Z 460.903,A -85,B 0,C 180,E1 -12461.611,E2 -12461.611} C_VEL
LIN {X 0,Y 375.963,Z 460.904,A -85,B 0,C 180,E1 -12465.262,E2 -12465.262} C_VEL
LIN {X 0,Y 375.974,Z 460.904,A -85,B 0,C 180,E1 -12469.139,E2 -12469.139} C_VEL
LIN {X 0,Y 375.962,Z 460.905,A -85,B 0,C 180,E1 -12471.912,E2 -12471.912} C_VEL
LIN {X 0,Y 375.974,Z 460.903,A -85,B 0,C 180,E1 -12475.333,E2 -12475.333} C_VEL
LIN {X 0,Y 375.952,Z 460.905,A -85,B 0,C 180,E1 -12478.438,E2 -12478.438} C_VEL
LIN {X 0,Y 375.979,Z 460.903,A -85,B 0,C 180,E1 -12482.141,E2 -12482.141} C_VEL
LIN {X 0,Y 376.012,Z 460.954,A -85,B 0,C 180,E1 -12485.426,E2 -12485.426} C_VEL
LIN {X 0,Y 376.191,Z 461.905,A -85,B 0,C 180,E1 -12486.263,E2 -12486.263} C_VEL
LIN {X 0,Y 377.537,Z 464.516,A -85,B 0,C 180,E1 -12487.386,E2 -12487.386} C_VEL
LIN {X 0,Y 379.169,Z 466.013,A -85,B 0,C 180,E1 -12488.527,E2 -12488.527} C_VEL
LIN {X 0,Y 381.534,Z 467.379,A -85,B 0,C 180,E1 -12490.216,E2 -12490.216} C_VEL
LIN {X 0,Y 383.697,Z 470.738,A -85,B 0,C 180,E1 -12492.062,E2 -12492.062} C_VEL
LIN {X 0,Y 385.739,Z 472.373,A -85,B 0,C 180,E1 -12493.869,E2 -12493.869} C_VEL
LIN {X 0,Y 387.794,Z 473.565,A -85,B 0,C 180,E1 -12495.839,E2 -12495.839} C_VEL
LIN {X 0,Y 389.572,Z 476.44,A -85,B 0,C 180,E1 -12498.027,E2 -12498.027} C_VEL
LIN {X 0,Y 391.109,Z 477.967,A -85,B 0,C 180,E1 -12500.133,E2 -12500.133} C_VEL
LIN {X 0,Y 392.714,Z 478.818,A -85,B 0,C 180,E1 -12502.804,E2 -12502.804} C_VEL
LIN {X 0,Y 393.622,Z 479.295,A -85,B 0,C 180,E1 -12504.878,E2 -12504.878} C_VEL
LIN {X 0,Y 394.219,Z 479.632,A -85,B 0,C 180,E1 -12506.934,E2 -12506.934} C_VEL
LIN {X 0,Y 394.501,Z 479.886,A -85,B 0,C 180,E1 -12508.979,E2 -12508.979} C_VEL
LIN {X 0,Y 394.501,Z 479.89,A -85,B 0,C 180,E1 -12511.021,E2 -12511.021} C_VEL
LIN {X 0,Y 394.181,Z 479.61,A -85,B 0,C 180,E1 -12513.207,E2 -12513.207} C_VEL
LIN {X 0,Y 393.621,Z 479.294,A -85,B 0,C 180,E1 -12515.122,E2 -12515.122} C_VEL
LIN {X 0,Y 392.469,Z 478.693,A -85,B 0,C 180,E1 -12517.647,E2 -12517.647} C_VEL
LIN {X 0,Y 390.932,Z 477.814,A -85,B 0,C 180,E1 -12520.114,E2 -12520.114} C_VEL
LIN {X 0,Y 389.389,Z 476.164,A -85,B 0,C 180,E1 -12522.244,E2 -12522.244} C_VEL
LIN {X 0,Y 387.793,Z 473.564,A -85,B 0,C 180,E1 -12524.161,E2 -12524.161} C_VEL
LIN {X 0,Y 384.923,Z 471.853,A -85,B 0,C 180,E1 -12526.848,E2 -12526.848} C_VEL
LIN {X 0,Y 382.986,Z 469.856,A -85,B 0,C 180,E1 -12528.523,E2 -12528.523} C_VEL
LIN {X 0,Y 381.314,Z 467.139,A -85,B 0,C 180,E1 -12529.954,E2 -12529.954} C_VEL
LIN {X 0,Y 378.221,Z 465.275,A -85,B 0,C 180,E1 -12532.153,E2 -12532.153} C_VEL
LIN {X 0,Y 376.568,Z 462.936,A -85,B 0,C 180,E1 -12533.346,E2 -12533.346} C_VEL
LIN {X 0,Y 376.082,Z 461.437,A -85,B 0,C 180,E1 -12534,E2 -12534} C_VEL
LIN {X 0,Y 376.007,Z 460.927,A -85,B 0,C 180,E1 -12534.869,E2 -12534.869} C_VEL
LIN {X 0,Y 375.979,Z 460.904,A -85,B 0,C 180,E1 -12537.859,E2 -12537.859} C_VEL
LIN {X 0,Y 375.952,Z 460.905,A -85,B 0,C 180,E1 -12541.562,E2 -12541.562} C_VEL
LIN {X 0,Y 375.953,Z 460.904,A -85,B 0,C 180,E1 -12545.415,E2 -12545.415} C_VEL
LIN {X 0,Y 375.972,Z 460.903,A -85,B 0,C 180,E1 -12548.271,E2 -12548.271} C_VEL
LIN {X 0,Y 375.987,Z 460.9,A -85,B 0,C 180,E1 -12550.041,E2 -12550.041} C_VEL
LIN {X 0,Y 375.275,Z 460.99,A -85,B 0,C 180,E1 -12550.934,E2 -12550.934} C_VEL
LIN {X 0,Y 372.371,Z 461.353,A -85,B 0,C 180,E1 -12552.386,E2 -12552.386} C_VEL
LIN {X 0,Y 369.962,Z 461.652,A -85,B 0,C 180,E1 -12553.561,E2 -12553.561} C_VEL
LIN {X 0,Y 368.973,Z 461.774,A -85,B 0,C 180,E1 -12554.47,E2 -12554.47} C_VEL
LIN {X 0,Y 368.914,Z 461.782,A -85,B 0,C 180,E1 -12554.777,E2 -12554.777} C_VEL
LIN {X 0,Y 368.934,Z 461.781,A -85,B 0,C 180,E1 -12558.185,E2 -12558.185} C_VEL
LIN {X 0,Y 368.91,Z 461.784,A -85,B 0,C 180,E1 -12561.358,E2 -12561.358} C_VEL
LIN {X 0,Y 368.929,Z 461.737,A -85,B 0,C 180,E1 -12565.146,E2 -12565.146} C_VEL
LIN {X 0,Y 368.922,Z 461.78,A -85,B 0,C 180,E1 -12569.046,E2 -12569.046} C_VEL
LIN {X 0,Y 368.979,Z 461.742,A -85,B 0,C 180,E1 -12571.564,E2 -12571.564} C_VEL
LIN {X 0,Y 368.992,Z 461.722,A -85,B 0,C 180,E1 -12574.02,E2 -12574.02} C_VEL
LIN {X 0,Y 368.917,Z 461.781,A -85,B 0,C 180,E1 -12577.604,E2 -12577.604} C_VEL
LIN {X 0,Y 368.958,Z 461.772,A -85,B 0,C 180,E1 -12581.106,E2 -12581.106} C_VEL
LIN {X 0,Y 368.989,Z 461.755,A -85,B 0,C 180,E1 -12584.535,E2 -12584.535} C_VEL
LIN {X 0,Y 368.997,Z 461.758,A -85,B 0,C 180,E1 -12587.907,E2 -12587.907} C_VEL
LIN {X 0,Y 369.18,Z 461.743,A -85,B 0,C 180,E1 -12591.845,E2 -12591.845} C_VEL
LIN {X 0,Y 369.137,Z 461.742,A -85,B 0,C 180,E1 -12594.538,E2 -12594.538} C_VEL
LIN {X 0,Y 369.311,Z 461.717,A -85,B 0,C 180,E1 -12597.819,E2 -12597.819} C_VEL
LIN {X 0,Y 369.45,Z 461.71,A -85,B 0,C 180,E1 -12600,E2 -12600} C_VEL
LIN {X 0,Y 369.311,Z 461.726,A -85,B 0,C 180,E1 -12602.181,E2 -12602.181} C_VEL
LIN {X 0,Y 369.197,Z 461.743,A -85,B 0,C 180,E1 -12606.559,E2 -12606.559} C_VEL
LIN {X 0,Y 369.06,Z 461.754,A -85,B 0,C 180,E1 -12609.869,E2 -12609.869} C_VEL
LIN {X 0,Y 369.03,Z 461.752,A -85,B 0,C 180,E1 -12613.773,E2 -12613.773} C_VEL
LIN {X 0,Y 368.994,Z 461.745,A -85,B 0,C 180,E1 -12617.769,E2 -12617.769} C_VEL
LIN {X 0,Y 368.903,Z 461.731,A -85,B 0,C 180,E1 -12621.221,E2 -12621.221} C_VEL
LIN {X 0,Y 368.949,Z 461.776,A -85,B 0,C 180,E1 -12624.776,E2 -12624.776} C_VEL
LIN {X 0,Y 368.964,Z 461.733,A -85,B 0,C 180,E1 -12627.203,E2 -12627.203} C_VEL
LIN {X 0,Y 368.917,Z 461.743,A -85,B 0,C 180,E1 -12629.69,E2 -12629.69} C_VEL
LIN {X 0,Y 368.893,Z 461.765,A -85,B 0,C 180,E1 -12633.538,E2 -12633.538} C_VEL
LIN {X 0,Y 368.898,Z 461.776,A -85,B 0,C 180,E1 -12636.857,E2 -12636.857} C_VEL
LIN {X 0,Y 368.948,Z 461.754,A -85,B 0,C 180,E1 -12640.365,E2 -12640.365} C_VEL
LIN {X 0,Y 368.926,Z 461.762,A -85,B 0,C 180,E1 -12643.624,E2 -12643.624} C_VEL
LIN {X 0,Y 368.913,Z 461.833,A -85,B 0,C 180,E1 -12645.574,E2 -12645.574} C_VEL
LIN {X 0,Y 369.771,Z 464.79,A -85,B 0,C 180,E1 -12646.527,E2 -12646.527} C_VEL
LIN {X 0,Y 373.501,Z 477.394,A -85,B 0,C 180,E1 -12650.052,E2 -12650.052} C_VEL
LIN {X 0,Y 374.049,Z 478.924,A -85,B 0,C 180,E1 -12650.287,E2 -12650.287} C_VEL
LIN {X 0,Y 383.755,Z 496.893,A -85,B 0,C 180,E1 -12651.899,E2 -12651.899} C_VEL
LIN {X 0,Y 393.108,Z 516.212,A -85,B 0,C 180,E1 -12653.383,E2 -12653.383} C_VEL
LIN {X 0,Y 396.548,Z 531.373,A -85,B 0,C 180,E1 -12654.081,E2 -12654.081} C_VEL
LIN {X 0,Y 392.785,Z 660.791,A -85,B 0,C 180,E1 -12656.505,E2 -12656.505} C_VEL
LIN {X 0,Y 391.725,Z 692.702,A -85,B 0,C 180,E1 -12657.132,E2 -12657.132} C_VEL
LIN {X 0,Y 390.717,Z 707.341,A -85,B 0,C 180,E1 -12657.541,E2 -12657.541} C_VEL
LIN {X 0,Y 389.223,Z 724.632,A -85,B 0,C 180,E1 -12658.229,E2 -12658.229} C_VEL
LIN {X 0,Y 387.395,Z 740.611,A -85,B 0,C 180,E1 -12659.094,E2 -12659.094} C_VEL
LIN {X 0,Y 385.805,Z 753.253,A -85,B 0,C 180,E1 -12659.938,E2 -12659.938} C_VEL
LIN {X 0,Y 384.043,Z 764.893,A -85,B 0,C 180,E1 -12660.842,E2 -12660.842} C_VEL
LIN {X 0,Y 381.983,Z 777.747,A -85,B 0,C 180,E1 -12662.023,E2 -12662.023} C_VEL
LIN {X 0,Y 380.158,Z 788.865,A -85,B 0,C 180,E1 -12663.217,E2 -12663.217} C_VEL
LIN {X 0,Y 378.156,Z 799.706,A -85,B 0,C 180,E1 -12664.547,E2 -12664.547} C_VEL
LIN {X 0,Y 376.357,Z 809.713,A -85,B 0,C 180,E1 -12665.962,E2 -12665.962} C_VEL
LIN {X 0,Y 374.808,Z 818.607,A -85,B 0,C 180,E1 -12667.394,E2 -12667.394} C_VEL
LIN {X 0,Y 373.116,Z 827.566,A -85,B 0,C 180,E1 -12669.03,E2 -12669.03} C_VEL
LIN {X 0,Y 371.73,Z 835.703,A -85,B 0,C 180,E1 -12670.737,E2 -12670.737} C_VEL
LIN {X 0,Y 370.68,Z 842.428,A -85,B 0,C 180,E1 -12672.341,E2 -12672.341} C_VEL
LIN {X 0,Y 369.694,Z 848.568,A -85,B 0,C 180,E1 -12674,E2 -12674} C_VEL
LIN {X 0,Y 368.798,Z 855.474,A -85,B 0,C 180,E1 -12676.205,E2 -12676.205} C_VEL
LIN {X 0,Y 368.234,Z 859.983,A -85,B 0,C 180,E1 -12677.881,E2 -12677.881} C_VEL
LIN {X 0,Y 367.726,Z 864.878,A -85,B 0,C 180,E1 -12680.096,E2 -12680.096} C_VEL
LIN {X 0,Y 367.545,Z 868.727,A -85,B 0,C 180,E1 -12682.308,E2 -12682.308} C_VEL
LIN {X 0,Y 367.42,Z 871.572,A -85,B 0,C 180,E1 -12684.512,E2 -12684.512} C_VEL
LIN {X 0,Y 367.394,Z 872.705,A -85,B 0,C 180,E1 -12685.612,E2 -12685.612} C_VEL
LIN {X 0,Y 367.347,Z 874.124,A -85,B 0,C 180,E1 -12687.807,E2 -12687.807} C_VEL
LIN {X 0,Y 367.392,Z 874.597,A -85,B 0,C 180,E1 -12690,E2 -12690} C_VEL
LIN {X 0,Y 367.347,Z 874.124,A -85,B 0,C 180,E1 -12692.193,E2 -12692.193} C_VEL
LIN {X 0,Y 367.394,Z 872.705,A -85,B 0,C 180,E1 -12694.388,E2 -12694.388} C_VEL
LIN {X 0,Y 367.478,Z 870.326,A -85,B 0,C 180,E1 -12696.589,E2 -12696.589} C_VEL
LIN {X 0,Y 367.683,Z 865.918,A -85,B 0,C 180,E1 -12699.35,E2 -12699.35} C_VEL
LIN {X 0,Y 367.957,Z 862.554,A -85,B 0,C 180,E1 -12701.011,E2 -12701.011} C_VEL
LIN {X 0,Y 368.559,Z 857.058,A -85,B 0,C 180,E1 -12703.228,E2 -12703.228} C_VEL
LIN {X 0,Y 369.202,Z 852.201,A -85,B 0,C 180,E1 -12704.891,E2 -12704.891} C_VEL
LIN {X 0,Y 370.362,Z 844.535,A -85,B 0,C 180,E1 -12707.105,E2 -12707.105} C_VEL
LIN {X 0,Y 371.492,Z 837.158,A -85,B 0,C 180,E1 -12708.931,E2 -12708.931} C_VEL
LIN {X 0,Y 372.604,Z 830.324,A -85,B 0,C 180,E1 -12710.422,E2 -12710.422} C_VEL
LIN {X 0,Y 374.181,Z 821.739,A -85,B 0,C 180,E1 -12712.064,E2 -12712.064} C_VEL
LIN {X 0,Y 375.9,Z 812.352,A -85,B 0,C 180,E1 -12713.634,E2 -12713.634} C_VEL
LIN {X 0,Y 377.815,Z 801.721,A -85,B 0,C 180,E1 -12715.183,E2 -12715.183} C_VEL
LIN {X 0,Y 379.473,Z 792.295,A -85,B 0,C 180,E1 -12716.39,E2 -12716.39} C_VEL
LIN {X 0,Y 381.386,Z 781.524,A -85,B 0,C 180,E1 -12717.593,E2 -12717.593} C_VEL
LIN {X 0,Y 383.313,Z 769.394,A -85,B 0,C 180,E1 -12718.769,E2 -12718.769} C_VEL
LIN {X 0,Y 385.223,Z 756.734,A -85,B 0,C 180,E1 -12719.811,E2 -12719.811} C_VEL
LIN {X 0,Y 386.863,Z 744.715,A -85,B 0,C 180,E1 -12720.65,E2 -12720.65} C_VEL
LIN {X 0,Y 388.456,Z 731.507,A -85,B 0,C 180,E1 -12721.417,E2 -12721.417} C_VEL
LIN {X 0,Y 389.865,Z 717.814,A -85,B 0,C 180,E1 -12722.058,E2 -12722.058} C_VEL
LIN {X 0,Y 390.95,Z 705.222,A -85,B 0,C 180,E1 -12722.518,E2 -12722.518} C_VEL
LIN {X 0,Y 391.733,Z 692.703,A -85,B 0,C 180,E1 -12722.867,E2 -12722.867} C_VEL
LIN {X 0,Y 392.903,Z 657.209,A -85,B 0,C 180,E1 -12723.561,E2 -12723.561} C_VEL
LIN {X 0,Y 396.561,Z 531.435,A -85,B 0,C 180,E1 -12725.916,E2 -12725.916} C_VEL
LIN {X 0,Y 392.911,Z 515.759,A -85,B 0,C 180,E1 -12726.648,E2 -12726.648} C_VEL
LIN {X 0,Y 383.304,Z 495.971,A -85,B 0,C 180,E1 -12728.175,E2 -12728.175} C_VEL
LIN {X 0,Y 374.882,Z 480.613,A -85,B 0,C 180,E1 -12729.558,E2 -12729.558} C_VEL
LIN {X 0,Y 373.647,Z 477.932,A -85,B 0,C 180,E1 -12729.831,E2 -12729.831} C_VEL
LIN {X 0,Y 370.156,Z 466.007,A -85,B 0,C 180,E1 -12733.118,E2 -12733.118} C_VEL
LIN {X 0,Y 368.978,Z 462.114,A -85,B 0,C 180,E1 -12734.277,E2 -12734.277} C_VEL
LIN {X 0,Y 368.919,Z 461.768,A -85,B 0,C 180,E1 -12734.817,E2 -12734.817} C_VEL
LIN {X 0,Y 368.941,Z 461.776,A -85,B 0,C 180,E1 -12738.186,E2 -12738.186} C_VEL
LIN {X 0,Y 368.908,Z 461.771,A -85,B 0,C 180,E1 -12741.358,E2 -12741.358} C_VEL
LIN {X 0,Y 368.931,Z 461.747,A -85,B 0,C 180,E1 -12745.146,E2 -12745.146} C_VEL
LIN {X 0,Y 368.923,Z 461.771,A -85,B 0,C 180,E1 -12749.046,E2 -12749.046} C_VEL
LIN {X 0,Y 368.98,Z 461.722,A -85,B 0,C 180,E1 -12751.564,E2 -12751.564} C_VEL
LIN {X 0,Y 368.993,Z 461.754,A -85,B 0,C 180,E1 -12754.019,E2 -12754.019} C_VEL
LIN {X 0,Y 368.917,Z 461.754,A -85,B 0,C 180,E1 -12757.604,E2 -12757.604} C_VEL
LIN {X 0,Y 368.959,Z 461.725,A -85,B 0,C 180,E1 -12761.106,E2 -12761.106} C_VEL
LIN {X 0,Y 368.99,Z 461.77,A -85,B 0,C 180,E1 -12764.535,E2 -12764.535} C_VEL
LIN {X 0,Y 368.998,Z 461.762,A -85,B 0,C 180,E1 -12767.906,E2 -12767.906} C_VEL
LIN {X 0,Y 369.158,Z 461.733,A -85,B 0,C 180,E1 -12771.869,E2 -12771.869} C_VEL
LIN {X 0,Y 369.139,Z 461.751,A -85,B 0,C 180,E1 -12774.537,E2 -12774.537} C_VEL
LIN {X 0,Y 369.311,Z 461.725,A -85,B 0,C 180,E1 -12777.819,E2 -12777.819} C_VEL
LIN {X 0,Y 369.45,Z 461.708,A -85,B 0,C 180,E1 -12780,E2 -12780} C_VEL
LIN {X 0,Y 369.311,Z 461.714,A -85,B 0,C 180,E1 -12782.181,E2 -12782.181} C_VEL
LIN {X 0,Y 369.192,Z 461.728,A -85,B 0,C 180,E1 -12786.574,E2 -12786.574} C_VEL
LIN {X 0,Y 369.113,Z 461.755,A -85,B 0,C 180,E1 -12788.761,E2 -12788.761} C_VEL
LIN {X 0,Y 368.997,Z 461.758,A -85,B 0,C 180,E1 -12792.093,E2 -12792.093} C_VEL
LIN {X 0,Y 368.989,Z 461.755,A -85,B 0,C 180,E1 -12795.465,E2 -12795.465} C_VEL
LIN {X 0,Y 368.958,Z 461.773,A -85,B 0,C 180,E1 -12798.894,E2 -12798.894} C_VEL
LIN {X 0,Y 368.917,Z 461.781,A -85,B 0,C 180,E1 -12802.396,E2 -12802.396} C_VEL
LIN {X 0,Y 368.992,Z 461.722,A -85,B 0,C 180,E1 -12805.98,E2 -12805.98} C_VEL
LIN {X 0,Y 368.96,Z 461.755,A -85,B 0,C 180,E1 -12808.813,E2 -12808.813} C_VEL
LIN {X 0,Y 368.892,Z 461.76,A -85,B 0,C 180,E1 -12812.238,E2 -12812.238} C_VEL
LIN {X 0,Y 368.922,Z 461.74,A -85,B 0,C 180,E1 -12815.002,E2 -12815.002} C_VEL
LIN {X 0,Y 368.91,Z 461.784,A -85,B 0,C 180,E1 -12818.642,E2 -12818.642} C_VEL
LIN {X 0,Y 368.935,Z 461.78,A -85,B 0,C 180,E1 -12822.02,E2 -12822.02} C_VEL
LIN {X 0,Y 368.918,Z 461.782,A -85,B 0,C 180,E1 -12825.183,E2 -12825.183} C_VEL
LIN {X 0,Y 368.904,Z 461.783,A -85,B 0,C 180,E1 -12828.182,E2 -12828.182} C_VEL
LIN {X 0,Y 368.907,Z 461.782,A -85,B 0,C 180,E1 -12831.359,E2 -12831.359} C_VEL
LIN {X 0,Y 368.931,Z 461.782,A -85,B 0,C 180,E1 -12835.147,E2 -12835.147} C_VEL
LIN {X 0,Y 368.924,Z 461.781,A -85,B 0,C 180,E1 -12839.047,E2 -12839.047} C_VEL
LIN {X 0,Y 368.952,Z 461.909,A -85,B 0,C 180,E1 -12841.872,E2 -12841.872} C_VEL
LIN {X 0,Y 369.278,Z 463.208,A -85,B 0,C 180,E1 -12842.631,E2 -12842.631} C_VEL
LIN {X 0,Y 370.611,Z 465.492,A -85,B 0,C 180,E1 -12843.506,E2 -12843.506} C_VEL
LIN {X 0,Y 373.112,Z 467.403,A -85,B 0,C 180,E1 -12844.999,E2 -12844.999} C_VEL
LIN {X 0,Y 374.56,Z 468.426,A -85,B 0,C 180,E1 -12845.912,E2 -12845.912} C_VEL
LIN {X 0,Y 376.249,Z 471.292,A -85,B 0,C 180,E1 -12847.123,E2 -12847.123} C_VEL
LIN {X 0,Y 378.194,Z 473.043,A -85,B 0,C 180,E1 -12848.469,E2 -12848.469} C_VEL
LIN {X 0,Y 380.467,Z 474.354,A -85,B 0,C 180,E1 -12850.086,E2 -12850.086} C_VEL
LIN {X 0,Y 382.291,Z 477.327,A -85,B 0,C 180,E1 -12851.65,E2 -12851.65} C_VEL
LIN {X 0,Y 384.516,Z 479.221,A -85,B 0,C 180,E1 -12853.543,E2 -12853.543} C_VEL
LIN {X 0,Y 386.878,Z 480.636,A -85,B 0,C 180,E1 -12855.804,E2 -12855.804} C_VEL
LIN {X 0,Y 388.58,Z 483.384,A -85,B 0,C 180,E1 -12857.863,E2 -12857.863} C_VEL
LIN {X 0,Y 390.22,Z 485.012,A -85,B 0,C 180,E1 -12860.11,E2 -12860.11} C_VEL
LIN {X 0,Y 391.838,Z 485.855,A -85,B 0,C 180,E1 -12862.788,E2 -12862.788} C_VEL
LIN {X 0,Y 392.753,Z 486.344,A -85,B 0,C 180,E1 -12864.867,E2 -12864.867} C_VEL
LIN {X 0,Y 393.352,Z 486.678,A -85,B 0,C 180,E1 -12866.928,E2 -12866.928} C_VEL
LIN {X 0,Y 393.637,Z 486.92,A -85,B 0,C 180,E1 -12868.977,E2 -12868.977} C_VEL
LIN {X 0,Y 393.64,Z 486.901,A -85,B 0,C 180,E1 -12871.126,E2 -12871.126} C_VEL
LIN {X 0,Y 393.353,Z 486.678,A -85,B 0,C 180,E1 -12873.072,E2 -12873.072} C_VEL
LIN {X 0,Y 392.751,Z 486.343,A -85,B 0,C 180,E1 -12875.133,E2 -12875.133} C_VEL
LIN {X 0,Y 391.593,Z 485.737,A -85,B 0,C 180,E1 -12877.664,E2 -12877.664} C_VEL
LIN {X 0,Y 390.044,Z 484.861,A -85,B 0,C 180,E1 -12880.137,E2 -12880.137} C_VEL
LIN {X 0,Y 388.454,Z 483.178,A -85,B 0,C 180,E1 -12882.32,E2 -12882.32} C_VEL
LIN {X 0,Y 386.614,Z 480.335,A -85,B 0,C 180,E1 -12884.474,E2 -12884.474} C_VEL
LIN {X 0,Y 383.82,Z 478.76,A -85,B 0,C 180,E1 -12887.035,E2 -12887.035} C_VEL
LIN {X 0,Y 381.863,Z 476.726,A -85,B 0,C 180,E1 -12888.719,E2 -12888.719} C_VEL
LIN {X 0,Y 380.176,Z 474.032,A -85,B 0,C 180,E1 -12890.143,E2 -12890.143} C_VEL
LIN {X 0,Y 377.182,Z 472.31,A -85,B 0,C 180,E1 -12892.239,E2 -12892.239} C_VEL
LIN {X 0,Y 375.262,Z 469.781,A -85,B 0,C 180,E1 -12893.597,E2 -12893.597} C_VEL
LIN {X 0,Y 374.271,Z 468.1,A -85,B 0,C 180,E1 -12894.283,E2 -12894.283} C_VEL
LIN {X 0,Y 370.911,Z 465.817,A -85,B 0,C 180,E1 -12896.324,E2 -12896.324} C_VEL
LIN {X 0,Y 369.331,Z 463.375,A -85,B 0,C 180,E1 -12897.327,E2 -12897.327} C_VEL
LIN {X 0,Y 369.023,Z 462.284,A -85,B 0,C 180,E1 -12897.813,E2 -12897.813} C_VEL
LIN {X 0,Y 368.958,Z 461.813,A -85,B 0,C 180,E1 -12898.437,E2 -12898.437} C_VEL
LIN {X 0,Y 368.893,Z 461.785,A -85,B 0,C 180,E1 -12902.238,E2 -12902.238} C_VEL
LIN {X 0,Y 368.924,Z 461.782,A -85,B 0,C 180,E1 -12905.001,E2 -12905.001} C_VEL
LIN {X 0,Y 368.907,Z 461.782,A -85,B 0,C 180,E1 -12908.641,E2 -12908.641} C_VEL
LIN {X 0,Y 368.904,Z 461.783,A -85,B 0,C 180,E1 -12911.818,E2 -12911.818} C_VEL
LIN {X 0,Y 368.914,Z 461.782,A -85,B 0,C 180,E1 -12914.777,E2 -12914.777} C_VEL
LIN {X 0,Y 368.308,Z 461.863,A -85,B 0,C 180,E1 -12915.688,E2 -12915.688} C_VEL
LIN {X 0,Y 365.477,Z 462.216,A -85,B 0,C 180,E1 -12917.17,E2 -12917.17} C_VEL
LIN {X 0,Y 363.034,Z 462.517,A -85,B 0,C 180,E1 -12918.368,E2 -12918.368} C_VEL
LIN {X 0,Y 361.97,Z 462.648,A -85,B 0,C 180,E1 -12919.295,E2 -12919.295} C_VEL
LIN {X 0,Y 361.878,Z 462.658,A -85,B 0,C 180,E1 -12919.609,E2 -12919.609} C_VEL
LIN {X 0,Y 361.87,Z 462.659,A -85,B 0,C 180,E1 -12922.983,E2 -12922.983} C_VEL
LIN {X 0,Y 361.851,Z 462.616,A -85,B 0,C 180,E1 -12926.631,E2 -12926.631} C_VEL
LIN {X 0,Y 361.869,Z 462.659,A -85,B 0,C 180,E1 -12929.672,E2 -12929.672} C_VEL
LIN {X 0,Y 361.947,Z 462.595,A -85,B 0,C 180,E1 -12933.475,E2 -12933.475} C_VEL
LIN {X 0,Y 361.874,Z 462.659,A -85,B 0,C 180,E1 -12937.144,E2 -12937.144} C_VEL
LIN {X 0,Y 361.901,Z 462.647,A -85,B 0,C 180,E1 -12940.723,E2 -12940.723} C_VEL
LIN {X 0,Y 361.924,Z 462.642,A -85,B 0,C 180,E1 -12943.066,E2 -12943.066} C_VEL
LIN {X 0,Y 361.991,Z 462.641,A -85,B 0,C 180,E1 -12946.528,E2 -12946.528} C_VEL
LIN {X 0,Y 362.023,Z 462.63,A -85,B 0,C 180,E1 -12949.938,E2 -12949.938} C_VEL
LIN {X 0,Y 362.155,Z 462.606,A -85,B 0,C 180,E1 -12953.314,E2 -12953.314} C_VEL
LIN {X 0,Y 362.275,Z 462.593,A -85,B 0,C 180,E1 -12957.777,E2 -12957.777} C_VEL
LIN {X 0,Y 362.419,Z 462.585,A -85,B 0,C 180,E1 -12960,E2 -12960} C_VEL
LIN {X 0,Y 362.275,Z 462.602,A -85,B 0,C 180,E1 -12962.224,E2 -12962.224} C_VEL
LIN {X 0,Y 362.158,Z 462.62,A -85,B 0,C 180,E1 -12966.687,E2 -12966.687} C_VEL
LIN {X 0,Y 362.024,Z 462.634,A -85,B 0,C 180,E1 -12970.062,E2 -12970.062} C_VEL
LIN {X 0,Y 361.99,Z 462.629,A -85,B 0,C 180,E1 -12973.899,E2 -12973.899} C_VEL
LIN {X 0,Y 361.96,Z 462.617,A -85,B 0,C 180,E1 -12977.939,E2 -12977.939} C_VEL
LIN {X 0,Y 361.855,Z 462.615,A -85,B 0,C 180,E1 -12981.655,E2 -12981.655} C_VEL
LIN {X 0,Y 361.92,Z 462.648,A -85,B 0,C 180,E1 -12985.291,E2 -12985.291} C_VEL
LIN {X 0,Y 361.916,Z 462.603,A -85,B 0,C 180,E1 -12987.778,E2 -12987.778} C_VEL
LIN {X 0,Y 361.854,Z 462.66,A -85,B 0,C 180,E1 -12991.628,E2 -12991.628} C_VEL
LIN {X 0,Y 361.869,Z 462.627,A -85,B 0,C 180,E1 -12995.345,E2 -12995.345} C_VEL
LIN {X 0,Y 361.869,Z 462.641,A -85,B 0,C 180,E1 -12999.028,E2 -12999.028} C_VEL
LIN {X 0,Y 361.884,Z 462.658,A -85,B 0,C 180,E1 -13002.442,E2 -13002.442} C_VEL
LIN {X 0,Y 361.931,Z 462.769,A -85,B 0,C 180,E1 -13004.829,E2 -13004.829} C_VEL
LIN {X 0,Y 364.555,Z 471.758,A -85,B 0,C 180,E1 -13007.567,E2 -13007.567} C_VEL
LIN {X 0,Y 366.362,Z 477.766,A -85,B 0,C 180,E1 -13009.234,E2 -13009.234} C_VEL
LIN {X 0,Y 374.607,Z 492.862,A -85,B 0,C 180,E1 -13010.704,E2 -13010.704} C_VEL
LIN {X 0,Y 383.135,Z 509.579,A -85,B 0,C 180,E1 -13012.122,E2 -13012.122} C_VEL
LIN {X 0,Y 387.805,Z 519.657,A -85,B 0,C 180,E1 -13012.881,E2 -13012.881} C_VEL
LIN {X 0,Y 390.765,Z 532.72,A -85,B 0,C 180,E1 -13013.499,E2 -13013.499} C_VEL
LIN {X 0,Y 386.893,Z 660.581,A -85,B 0,C 180,E1 -13015.926,E2 -13015.926} C_VEL
LIN {X 0,Y 385.783,Z 692.493,A -85,B 0,C 180,E1 -13016.56,E2 -13016.56} C_VEL
LIN {X 0,Y 384.755,Z 706.933,A -85,B 0,C 180,E1 -13016.967,E2 -13016.967} C_VEL
LIN {X 0,Y 383.194,Z 724.242,A -85,B 0,C 180,E1 -13017.658,E2 -13017.658} C_VEL
LIN {X 0,Y 381.289,Z 740.4,A -85,B 0,C 180,E1 -13018.544,E2 -13018.544} C_VEL
LIN {X 0,Y 379.627,Z 753.041,A -85,B 0,C 180,E1 -13019.397,E2 -13019.397} C_VEL
LIN {X 0,Y 377.826,Z 764.683,A -85,B 0,C 180,E1 -13020.314,E2 -13020.314} C_VEL
LIN {X 0,Y 375.883,Z 776.478,A -85,B 0,C 180,E1 -13021.404,E2 -13021.404} C_VEL
LIN {X 0,Y 373.94,Z 787.508,A -85,B 0,C 180,E1 -13022.584,E2 -13022.584} C_VEL
LIN {X 0,Y 371.833,Z 798.486,A -85,B 0,C 180,E1 -13023.932,E2 -13023.932} C_VEL
LIN {X 0,Y 370.022,Z 808.18,A -85,B 0,C 180,E1 -13025.301,E2 -13025.301} C_VEL
LIN {X 0,Y 368.156,Z 818.394,A -85,B 0,C 180,E1 -13026.963,E2 -13026.963} C_VEL
LIN {X 0,Y 366.361,Z 827.352,A -85,B 0,C 180,E1 -13028.625,E2 -13028.625} C_VEL
LIN {X 0,Y 364.888,Z 835.489,A -85,B 0,C 180,E1 -13030.361,E2 -13030.361} C_VEL
LIN {X 0,Y 363.806,Z 842.215,A -85,B 0,C 180,E1 -13031.996,E2 -13031.996} C_VEL
LIN {X 0,Y 362.772,Z 848.355,A -85,B 0,C 180,E1 -13033.686,E2 -13033.686} C_VEL
LIN {X 0,Y 361.772,Z 855.457,A -85,B 0,C 180,E1 -13036.004,E2 -13036.004} C_VEL
LIN {X 0,Y 361.069,Z 861.057,A -85,B 0,C 180,E1 -13038.207,E2 -13038.207} C_VEL
LIN {X 0,Y 360.655,Z 864.666,A -85,B 0,C 180,E1 -13039.899,E2 -13039.899} C_VEL
LIN {X 0,Y 360.462,Z 868.516,A -85,B 0,C 180,E1 -13042.156,E2 -13042.156} C_VEL
LIN {X 0,Y 360.33,Z 871.362,A -85,B 0,C 180,E1 -13044.404,E2 -13044.404} C_VEL
LIN {X 0,Y 360.307,Z 872.495,A -85,B 0,C 180,E1 -13045.525,E2 -13045.525} C_VEL
LIN {X 0,Y 360.251,Z 873.915,A -85,B 0,C 180,E1 -13047.764,E2 -13047.764} C_VEL
LIN {X 0,Y 360.296,Z 874.387,A -85,B 0,C 180,E1 -13050,E2 -13050} C_VEL
LIN {X 0,Y 360.251,Z 873.915,A -85,B 0,C 180,E1 -13052.236,E2 -13052.236} C_VEL
LIN {X 0,Y 360.307,Z 872.495,A -85,B 0,C 180,E1 -13054.475,E2 -13054.475} C_VEL
LIN {X 0,Y 360.382,Z 870.115,A -85,B 0,C 180,E1 -13056.719,E2 -13056.719} C_VEL
LIN {X 0,Y 360.598,Z 865.706,A -85,B 0,C 180,E1 -13059.536,E2 -13059.536} C_VEL
LIN {X 0,Y 360.902,Z 862.342,A -85,B 0,C 180,E1 -13061.229,E2 -13061.229} C_VEL
LIN {X 0,Y 361.646,Z 856.343,A -85,B 0,C 180,E1 -13063.672,E2 -13063.672} C_VEL
LIN {X 0,Y 362.231,Z 851.988,A -85,B 0,C 180,E1 -13065.184,E2 -13065.184} C_VEL
LIN {X 0,Y 363.484,Z 844.322,A -85,B 0,C 180,E1 -13067.439,E2 -13067.439} C_VEL
LIN {X 0,Y 364.565,Z 837.544,A -85,B 0,C 180,E1 -13069.16,E2 -13069.16} C_VEL
LIN {X 0,Y 365.862,Z 830.111,A -85,B 0,C 180,E1 -13070.816,E2 -13070.816} C_VEL
LIN {X 0,Y 367.51,Z 821.526,A -85,B 0,C 180,E1 -13072.486,E2 -13072.486} C_VEL
LIN {X 0,Y 369.414,Z 811.513,A -85,B 0,C 180,E1 -13074.18,E2 -13074.18} C_VEL
LIN {X 0,Y 371.428,Z 800.499,A -85,B 0,C 180,E1 -13075.797,E2 -13075.797} C_VEL
LIN {X 0,Y 373.263,Z 790.938,A -85,B 0,C 180,E1 -13077.015,E2 -13077.015} C_VEL
LIN {X 0,Y 375.25,Z 779.644,A -85,B 0,C 180,E1 -13078.278,E2 -13078.278} C_VEL
LIN {X 0,Y 377.057,Z 769.182,A -85,B 0,C 180,E1 -13079.292,E2 -13079.292} C_VEL
LIN {X 0,Y 379.033,Z 756.522,A -85,B 0,C 180,E1 -13080.348,E2 -13080.348} C_VEL
LIN {X 0,Y 380.751,Z 744.505,A -85,B 0,C 180,E1 -13081.196,E2 -13081.196} C_VEL
LIN {X 0,Y 382.399,Z 731.297,A -85,B 0,C 180,E1 -13081.973,E2 -13081.973} C_VEL
LIN {X 0,Y 383.755,Z 718.444,A -85,B 0,C 180,E1 -13082.589,E2 -13082.589} C_VEL
LIN {X 0,Y 384.961,Z 705.201,A -85,B 0,C 180,E1 -13083.081,E2 -13083.081} C_VEL
LIN {X 0,Y 385.783,Z 692.493,A -85,B 0,C 180,E1 -13083.44,E2 -13083.44} C_VEL
LIN {X 0,Y 386.945,Z 658.79,A -85,B 0,C 180,E1 -13084.109,E2 -13084.109} C_VEL
LIN {X 0,Y 390.805,Z 533.635,A -85,B 0,C 180,E1 -13086.476,E2 -13086.476} C_VEL
LIN {X 0,Y 388.965,Z 524.575,A -85,B 0,C 180,E1 -13086.879,E2 -13086.879} C_VEL
LIN {X 0,Y 387.354,Z 518.498,A -85,B 0,C 180,E1 -13087.195,E2 -13087.195} C_VEL
LIN {X 0,Y 378.343,Z 499.922,A -85,B 0,C 180,E1 -13088.67,E2 -13088.67} C_VEL
LIN {X 0,Y 368.687,Z 482.065,A -85,B 0,C 180,E1 -13090.316,E2 -13090.316} C_VEL
LIN {X 0,Y 366.27,Z 477.604,A -85,B 0,C 180,E1 -13090.8,E2 -13090.8} C_VEL
LIN {X 0,Y 363.14,Z 466.836,A -85,B 0,C 180,E1 -13093.87,E2 -13093.87} C_VEL
LIN {X 0,Y 361.932,Z 462.773,A -85,B 0,C 180,E1 -13095.168,E2 -13095.168} C_VEL
LIN {X 0,Y 361.901,Z 462.633,A -85,B 0,C 180,E1 -13099.231,E2 -13099.231} C_VEL
LIN {X 0,Y 361.868,Z 462.655,A -85,B 0,C 180,E1 -13102.982,E2 -13102.982} C_VEL
LIN {X 0,Y 361.856,Z 462.644,A -85,B 0,C 180,E1 -13106.629,E2 -13106.629} C_VEL
LIN {X 0,Y 361.871,Z 462.634,A -85,B 0,C 180,E1 -13109.672,E2 -13109.672} C_VEL
LIN {X 0,Y 361.948,Z 462.618,A -85,B 0,C 180,E1 -13113.475,E2 -13113.475} C_VEL
LIN {X 0,Y 361.875,Z 462.641,A -85,B 0,C 180,E1 -13117.144,E2 -13117.144} C_VEL
LIN {X 0,Y 361.902,Z 462.597,A -85,B 0,C 180,E1 -13120.723,E2 -13120.723} C_VEL
LIN {X 0,Y 361.925,Z 462.641,A -85,B 0,C 180,E1 -13123.066,E2 -13123.066} C_VEL
LIN {X 0,Y 361.991,Z 462.627,A -85,B 0,C 180,E1 -13126.527,E2 -13126.527} C_VEL
LIN {X 0,Y 362.024,Z 462.634,A -85,B 0,C 180,E1 -13129.938,E2 -13129.938} C_VEL
LIN {X 0,Y 362.158,Z 462.621,A -85,B 0,C 180,E1 -13133.313,E2 -13133.313} C_VEL
LIN {X 0,Y 362.275,Z 462.601,A -85,B 0,C 180,E1 -13137.776,E2 -13137.776} C_VEL
LIN {X 0,Y 362.419,Z 462.583,A -85,B 0,C 180,E1 -13140,E2 -13140} C_VEL
LIN {X 0,Y 362.275,Z 462.591,A -85,B 0,C 180,E1 -13142.223,E2 -13142.223} C_VEL
LIN {X 0,Y 362.155,Z 462.605,A -85,B 0,C 180,E1 -13146.686,E2 -13146.686} C_VEL
LIN {X 0,Y 362.023,Z 462.629,A -85,B 0,C 180,E1 -13150.062,E2 -13150.062} C_VEL
LIN {X 0,Y 361.99,Z 462.641,A -85,B 0,C 180,E1 -13153.899,E2 -13153.899} C_VEL
LIN {X 0,Y 361.96,Z 462.647,A -85,B 0,C 180,E1 -13157.939,E2 -13157.939} C_VEL
LIN {X 0,Y 361.873,Z 462.656,A -85,B 0,C 180,E1 -13161.654,E2 -13161.654} C_VEL
LIN {X 0,Y 361.919,Z 462.611,A -85,B 0,C 180,E1 -13165.29,E2 -13165.29} C_VEL
LIN {X 0,Y 361.915,Z 462.607,A -85,B 0,C 180,E1 -13167.778,E2 -13167.778} C_VEL
LIN {X 0,Y 361.84,Z 462.658,A -85,B 0,C 180,E1 -13171.285,E2 -13171.285} C_VEL
LIN {X 0,Y 361.847,Z 462.614,A -85,B 0,C 180,E1 -13174.281,E2 -13174.281} C_VEL
LIN {X 0,Y 361.869,Z 462.662,A -85,B 0,C 180,E1 -13177.226,E2 -13177.226} C_VEL
LIN {X 0,Y 361.899,Z 462.657,A -85,B 0,C 180,E1 -13180.768,E2 -13180.768} C_VEL
LIN {X 0,Y 361.905,Z 462.655,A -85,B 0,C 180,E1 -13184.354,E2 -13184.354} C_VEL
LIN {X 0,Y 361.851,Z 462.663,A -85,B 0,C 180,E1 -13187.565,E2 -13187.565} C_VEL
LIN {X 0,Y 361.869,Z 462.661,A -85,B 0,C 180,E1 -13190.973,E2 -13190.973} C_VEL
LIN {X 0,Y 361.869,Z 462.659,A -85,B 0,C 180,E1 -13194.655,E2 -13194.655} C_VEL
LIN {X 0,Y 361.876,Z 462.79,A -85,B 0,C 180,E1 -13198.514,E2 -13198.514} C_VEL
LIN {X 0,Y 362.225,Z 464.098,A -85,B 0,C 180,E1 -13199.218,E2 -13199.218} C_VEL
LIN {X 0,Y 363.362,Z 466.23,A -85,B 0,C 180,E1 -13199.91,E2 -13199.91} C_VEL
LIN {X 0,Y 365.487,Z 467.961,A -85,B 0,C 180,E1 -13201.036,E2 -13201.036} C_VEL
LIN {X 0,Y 367.327,Z 469.175,A -85,B 0,C 180,E1 -13202.047,E2 -13202.047} C_VEL
LIN {X 0,Y 369.231,Z 472.242,A -85,B 0,C 180,E1 -13203.241,E2 -13203.241} C_VEL
LIN {X 0,Y 371.504,Z 474.107,A -85,B 0,C 180,E1 -13204.595,E2 -13204.595} C_VEL
LIN {X 0,Y 373.245,Z 475.195,A -85,B 0,C 180,E1 -13205.646,E2 -13205.646} C_VEL
LIN {X 0,Y 375.024,Z 478.131,A -85,B 0,C 180,E1 -13206.898,E2 -13206.898} C_VEL
LIN {X 0,Y 377.068,Z 479.973,A -85,B 0,C 180,E1 -13208.301,E2 -13208.301} C_VEL
LIN {X 0,Y 379.357,Z 481.269,A -85,B 0,C 180,E1 -13209.918,E2 -13209.918} C_VEL
LIN {X 0,Y 381.164,Z 484.191,A -85,B 0,C 180,E1 -13211.455,E2 -13211.455} C_VEL
LIN {X 0,Y 383.59,Z 486.232,A -85,B 0,C 180,E1 -13213.502,E2 -13213.502} C_VEL
LIN {X 0,Y 385.83,Z 487.561,A -85,B 0,C 180,E1 -13215.63,E2 -13215.63} C_VEL
LIN {X 0,Y 387.645,Z 490.4,A -85,B 0,C 180,E1 -13217.778,E2 -13217.778} C_VEL
LIN {X 0,Y 389.332,Z 492.056,A -85,B 0,C 180,E1 -13220.087,E2 -13220.087} C_VEL
LIN {X 0,Y 390.962,Z 492.886,A -85,B 0,C 180,E1 -13222.771,E2 -13222.771} C_VEL
LIN {X 0,Y 391.883,Z 493.392,A -85,B 0,C 180,E1 -13224.856,E2 -13224.856} C_VEL
LIN {X 0,Y 392.487,Z 493.715,A -85,B 0,C 180,E1 -13226.921,E2 -13226.921} C_VEL
LIN {X 0,Y 392.772,Z 493.966,A -85,B 0,C 180,E1 -13228.975,E2 -13228.975} C_VEL
LIN {X 0,Y 392.772,Z 493.97,A -85,B 0,C 180,E1 -13231.025,E2 -13231.025} C_VEL
LIN {X 0,Y 392.487,Z 493.716,A -85,B 0,C 180,E1 -13233.079,E2 -13233.079} C_VEL
LIN {X 0,Y 391.882,Z 493.388,A -85,B 0,C 180,E1 -13235.144,E2 -13235.144} C_VEL
LIN {X 0,Y 390.717,Z 492.777,A -85,B 0,C 180,E1 -13237.681,E2 -13237.681} C_VEL
LIN {X 0,Y 389.159,Z 491.879,A -85,B 0,C 180,E1 -13240.161,E2 -13240.161} C_VEL
LIN {X 0,Y 387.473,Z 490.212,A -85,B 0,C 180,E1 -13242.424,E2 -13242.424} C_VEL
LIN {X 0,Y 385.57,Z 487.278,A -85,B 0,C 180,E1 -13244.649,E2 -13244.649} C_VEL
LIN {X 0,Y 382.886,Z 485.808,A -85,B 0,C 180,E1 -13247.078,E2 -13247.078} C_VEL
LIN {X 0,Y 380.74,Z 483.629,A -85,B 0,C 180,E1 -13248.916,E2 -13248.916} C_VEL
LIN {X 0,Y 379.067,Z 480.971,A -85,B 0,C 180,E1 -13250.312,E2 -13250.312} C_VEL
LIN {X 0,Y 376.061,Z 479.26,A -85,B 0,C 180,E1 -13252.381,E2 -13252.381} C_VEL
LIN {X 0,Y 374.054,Z 476.778,A -85,B 0,C 180,E1 -13253.775,E2 -13253.775} C_VEL
LIN {X 0,Y 372.937,Z 474.841,A -85,B 0,C 180,E1 -13254.567,E2 -13254.567} C_VEL
LIN {X 0,Y 369.847,Z 472.851,A -85,B 0,C 180,E1 -13256.406,E2 -13256.406} C_VEL
LIN {X 0,Y 367.994,Z 470.347,A -85,B 0,C 180,E1 -13257.55,E2 -13257.55} C_VEL
LIN {X 0,Y 366.87,Z 468.67,A -85,B 0,C 180,E1 -13258.213,E2 -13258.213} C_VEL
LIN {X 0,Y 364.074,Z 466.98,A -85,B 0,C 180,E1 -13259.697,E2 -13259.697} C_VEL
LIN {X 0,Y 362.503,Z 464.847,A -85,B 0,C 180,E1 -13260.593,E2 -13260.593} C_VEL
LIN {X 0,Y 361.996,Z 463.421,A -85,B 0,C 180,E1 -13261.047,E2 -13261.047} C_VEL
LIN {X 0,Y 361.864,Z 462.725,A -85,B 0,C 180,E1 -13261.626,E2 -13261.626} C_VEL
LIN {X 0,Y 361.869,Z 462.659,A -85,B 0,C 180,E1 -13265.345,E2 -13265.345} C_VEL
LIN {X 0,Y 361.869,Z 462.661,A -85,B 0,C 180,E1 -13269.027,E2 -13269.027} C_VEL
LIN {X 0,Y 361.851,Z 462.663,A -85,B 0,C 180,E1 -13272.435,E2 -13272.435} C_VEL
LIN {X 0,Y 361.906,Z 462.655,A -85,B 0,C 180,E1 -13275.931,E2 -13275.931} C_VEL
LIN {X 0,Y 361.878,Z 462.658,A -85,B 0,C 180,E1 -13279.609,E2 -13279.609} C_VEL
LIN {X 0,Y 361.197,Z 462.745,A -85,B 0,C 180,E1 -13280.537,E2 -13280.537} C_VEL
LIN {X 0,Y 358.346,Z 463.099,A -85,B 0,C 180,E1 -13282.047,E2 -13282.047} C_VEL
LIN {X 0,Y 355.935,Z 463.395,A -85,B 0,C 180,E1 -13283.269,E2 -13283.269} C_VEL
LIN {X 0,Y 354.895,Z 463.5,A -85,B 0,C 180,E1 -13284.214,E2 -13284.214} C_VEL
LIN {X 0,Y 354.806,Z 463.503,A -85,B 0,C 180,E1 -13284.534,E2 -13284.534} C_VEL
LIN {X 0,Y 354.78,Z 463.512,A -85,B 0,C 180,E1 -13287.666,E2 -13287.666} C_VEL
LIN {X 0,Y 354.862,Z 463.52,A -85,B 0,C 180,E1 -13290.621,E2 -13290.621} C_VEL
LIN {X 0,Y 354.891,Z 463.476,A -85,B 0,C 180,E1 -13294.172,E2 -13294.172} C_VEL
LIN {X 0,Y 354.819,Z 463.536,A -85,B 0,C 180,E1 -13297.893,E2 -13297.893} C_VEL
LIN {X 0,Y 354.915,Z 463.525,A -85,B 0,C 180,E1 -13301.892,E2 -13301.892} C_VEL
LIN {X 0,Y 354.935,Z 463.52,A -85,B 0,C 180,E1 -13305.981,E2 -13305.981} C_VEL
LIN {X 0,Y 354.97,Z 463.505,A -85,B 0,C 180,E1 -13309.736,E2 -13309.736} C_VEL
LIN {X 0,Y 355.12,Z 463.483,A -85,B 0,C 180,E1 -13313.181,E2 -13313.181} C_VEL
LIN {X 0,Y 355.238,Z 463.47,A -85,B 0,C 180,E1 -13317.733,E2 -13317.733} C_VEL
LIN {X 0,Y 355.368,Z 463.462,A -85,B 0,C 180,E1 -13320,E2 -13320} C_VEL
LIN {X 0,Y 355.238,Z 463.478,A -85,B 0,C 180,E1 -13322.268,E2 -13322.268} C_VEL
LIN {X 0,Y 355.121,Z 463.497,A -85,B 0,C 180,E1 -13326.82,E2 -13326.82} C_VEL
LIN {X 0,Y 354.971,Z 463.516,A -85,B 0,C 180,E1 -13330.264,E2 -13330.264} C_VEL
LIN {X 0,Y 354.935,Z 463.508,A -85,B 0,C 180,E1 -13334.019,E2 -13334.019} C_VEL
LIN {X 0,Y 354.916,Z 463.487,A -85,B 0,C 180,E1 -13338.109,E2 -13338.109} C_VEL
LIN {X 0,Y 354.81,Z 463.501,A -85,B 0,C 180,E1 -13342.108,E2 -13342.108} C_VEL
LIN {X 0,Y 354.892,Z 463.512,A -85,B 0,C 180,E1 -13345.828,E2 -13345.828} C_VEL
LIN {X 0,Y 354.849,Z 463.492,A -85,B 0,C 180,E1 -13349.679,E2 -13349.679} C_VEL
LIN {X 0,Y 354.825,Z 463.513,A -85,B 0,C 180,E1 -13353.683,E2 -13353.683} C_VEL
LIN {X 0,Y 354.796,Z 463.522,A -85,B 0,C 180,E1 -13356.46,E2 -13356.46} C_VEL
LIN {X 0,Y 354.819,Z 463.513,A -85,B 0,C 180,E1 -13359.424,E2 -13359.424} C_VEL
LIN {X 0,Y 354.831,Z 463.526,A -85,B 0,C 180,E1 -13362.876,E2 -13362.876} C_VEL
LIN {X 0,Y 354.88,Z 463.666,A -85,B 0,C 180,E1 -13364.016,E2 -13364.016} C_VEL
LIN {X 0,Y 357.741,Z 473.284,A -85,B 0,C 180,E1 -13367.037,E2 -13367.037} C_VEL
LIN {X 0,Y 359.031,Z 477.589,A -85,B 0,C 180,E1 -13368.233,E2 -13368.233} C_VEL
LIN {X 0,Y 365.517,Z 489.109,A -85,B 0,C 180,E1 -13369.442,E2 -13369.442} C_VEL
LIN {X 0,Y 374.598,Z 506.208,A -85,B 0,C 180,E1 -13371.025,E2 -13371.025} C_VEL
LIN {X 0,Y 382.455,Z 522.578,A -85,B 0,C 180,E1 -13372.345,E2 -13372.345} C_VEL
LIN {X 0,Y 385.057,Z 534.812,A -85,B 0,C 180,E1 -13372.921,E2 -13372.921} C_VEL
LIN {X 0,Y 380.384,Z 680.073,A -85,B 0,C 180,E1 -13375.701,E2 -13375.701} C_VEL
LIN {X 0,Y 379.422,Z 699.74,A -85,B 0,C 180,E1 -13376.163,E2 -13376.163} C_VEL
LIN {X 0,Y 378.124,Z 714.589,A -85,B 0,C 180,E1 -13376.675,E2 -13376.675} C_VEL
LIN {X 0,Y 376.647,Z 728.616,A -85,B 0,C 180,E1 -13377.32,E2 -13377.32} C_VEL
LIN {X 0,Y 375.075,Z 741.215,A -85,B 0,C 180,E1 -13378.04,E2 -13378.04} C_VEL
LIN {X 0,Y 373.462,Z 752.829,A -85,B 0,C 180,E1 -13378.836,E2 -13378.836} C_VEL
LIN {X 0,Y 371.608,Z 764.471,A -85,B 0,C 180,E1 -13379.766,E2 -13379.766} C_VEL
LIN {X 0,Y 369.509,Z 776.717,A -85,B 0,C 180,E1 -13380.918,E2 -13380.918} C_VEL
LIN {X 0,Y 367.568,Z 787.295,A -85,B 0,C 180,E1 -13382.067,E2 -13382.067} C_VEL
LIN {X 0,Y 365.382,Z 798.273,A -85,B 0,C 180,E1 -13383.436,E2 -13383.436} C_VEL
LIN {X 0,Y 363.48,Z 807.967,A -85,B 0,C 180,E1 -13384.826,E2 -13384.826} C_VEL
LIN {X 0,Y 361.515,Z 818.181,A -85,B 0,C 180,E1 -13386.514,E2 -13386.514} C_VEL
LIN {X 0,Y 359.668,Z 827.139,A -85,B 0,C 180,E1 -13388.207,E2 -13388.207} C_VEL
LIN {X 0,Y 358.134,Z 835.033,A -85,B 0,C 180,E1 -13389.915,E2 -13389.915} C_VEL
LIN {X 0,Y 356.912,Z 842,A -85,B 0,C 180,E1 -13391.636,E2 -13391.636} C_VEL
LIN {X 0,Y 355.845,Z 848.141,A -85,B 0,C 180,E1 -13393.359,E2 -13393.359} C_VEL
LIN {X 0,Y 354.79,Z 855.09,A -85,B 0,C 180,E1 -13395.665,E2 -13395.665} C_VEL
LIN {X 0,Y 354.206,Z 859.559,A -85,B 0,C 180,E1 -13397.394,E2 -13397.394} C_VEL
LIN {X 0,Y 353.598,Z 864.454,A -85,B 0,C 180,E1 -13399.696,E2 -13399.696} C_VEL
LIN {X 0,Y 353.373,Z 868.304,A -85,B 0,C 180,E1 -13401.998,E2 -13401.998} C_VEL
LIN {X 0,Y 353.26,Z 871.152,A -85,B 0,C 180,E1 -13404.291,E2 -13404.291} C_VEL
LIN {X 0,Y 353.222,Z 872.285,A -85,B 0,C 180,E1 -13405.435,E2 -13405.435} C_VEL
LIN {X 0,Y 353.159,Z 873.705,A -85,B 0,C 180,E1 -13407.719,E2 -13407.719} C_VEL
LIN {X 0,Y 353.199,Z 874.178,A -85,B 0,C 180,E1 -13410,E2 -13410} C_VEL
LIN {X 0,Y 353.159,Z 873.705,A -85,B 0,C 180,E1 -13412.281,E2 -13412.281} C_VEL
LIN {X 0,Y 353.222,Z 872.285,A -85,B 0,C 180,E1 -13414.565,E2 -13414.565} C_VEL
LIN {X 0,Y 353.298,Z 869.904,A -85,B 0,C 180,E1 -13416.855,E2 -13416.855} C_VEL
LIN {X 0,Y 353.528,Z 865.494,A -85,B 0,C 180,E1 -13419.728,E2 -13419.728} C_VEL
LIN {X 0,Y 353.864,Z 862.129,A -85,B 0,C 180,E1 -13421.455,E2 -13421.455} C_VEL
LIN {X 0,Y 354.585,Z 856.563,A -85,B 0,C 180,E1 -13423.786,E2 -13423.786} C_VEL
LIN {X 0,Y 355.267,Z 851.774,A -85,B 0,C 180,E1 -13425.489,E2 -13425.489} C_VEL
LIN {X 0,Y 356.612,Z 844.109,A -85,B 0,C 180,E1 -13427.786,E2 -13427.786} C_VEL
LIN {X 0,Y 357.713,Z 837.452,A -85,B 0,C 180,E1 -13429.511,E2 -13429.511} C_VEL
LIN {X 0,Y 359.124,Z 829.898,A -85,B 0,C 180,E1 -13431.225,E2 -13431.225} C_VEL
LIN {X 0,Y 360.884,Z 821.314,A -85,B 0,C 180,E1 -13432.922,E2 -13432.922} C_VEL
LIN {X 0,Y 362.77,Z 811.712,A -85,B 0,C 180,E1 -13434.582,E2 -13434.582} C_VEL
LIN {X 0,Y 364.761,Z 801.293,A -85,B 0,C 180,E1 -13436.151,E2 -13436.151} C_VEL
LIN {X 0,Y 366.908,Z 790.727,A -85,B 0,C 180,E1 -13437.522,E2 -13437.522} C_VEL
LIN {X 0,Y 368.761,Z 780.406,A -85,B 0,C 180,E1 -13438.706,E2 -13438.706} C_VEL
LIN {X 0,Y 370.829,Z 768.971,A -85,B 0,C 180,E1 -13439.834,E2 -13439.834} C_VEL
LIN {X 0,Y 372.615,Z 758.053,A -85,B 0,C 180,E1 -13440.771,E2 -13440.771} C_VEL
LIN {X 0,Y 374.656,Z 744.294,A -85,B 0,C 180,E1 -13441.762,E2 -13441.762} C_VEL
LIN {X 0,Y 376.348,Z 731.085,A -85,B 0,C 180,E1 -13442.55,E2 -13442.55} C_VEL
LIN {X 0,Y 377.787,Z 718.089,A -85,B 0,C 180,E1 -13443.177,E2 -13443.177} C_VEL
LIN {X 0,Y 378.995,Z 705.199,A -85,B 0,C 180,E1 -13443.662,E2 -13443.662} C_VEL
LIN {X 0,Y 379.876,Z 692.283,A -85,B 0,C 180,E1 -13444.031,E2 -13444.031} C_VEL
LIN {X 0,Y 381.153,Z 656.79,A -85,B 0,C 180,E1 -13444.74,E2 -13444.74} C_VEL
LIN {X 0,Y 385.026,Z 534.035,A -85,B 0,C 180,E1 -13447.101,E2 -13447.101} C_VEL
LIN {X 0,Y 382.31,Z 522.329,A -85,B 0,C 180,E1 -13447.678,E2 -13447.678} C_VEL
LIN {X 0,Y 373.711,Z 504.414,A -85,B 0,C 180,E1 -13449.127,E2 -13449.127} C_VEL
LIN {X 0,Y 364.067,Z 486.411,A -85,B 0,C 180,E1 -13450.82,E2 -13450.82} C_VEL
LIN {X 0,Y 358.927,Z 477.353,A -85,B 0,C 180,E1 -13451.806,E2 -13451.806} C_VEL
LIN {X 0,Y 356.022,Z 467.53,A -85,B 0,C 180,E1 -13454.712,E2 -13454.712} C_VEL
LIN {X 0,Y 354.88,Z 463.675,A -85,B 0,C 180,E1 -13455.984,E2 -13455.984} C_VEL
LIN {X 0,Y 354.853,Z 463.511,A -85,B 0,C 180,E1 -13459.188,E2 -13459.188} C_VEL
LIN {X 0,Y 354.808,Z 463.54,A -85,B 0,C 180,E1 -13462.401,E2 -13462.401} C_VEL
LIN {X 0,Y 354.807,Z 463.505,A -85,B 0,C 180,E1 -13464.94,E2 -13464.94} C_VEL
LIN {X 0,Y 354.809,Z 463.537,A -85,B 0,C 180,E1 -13468.399,E2 -13468.399} C_VEL
LIN {X 0,Y 354.847,Z 463.479,A -85,B 0,C 180,E1 -13471.619,E2 -13471.619} C_VEL
LIN {X 0,Y 354.892,Z 463.512,A -85,B 0,C 180,E1 -13474.172,E2 -13474.172} C_VEL
LIN {X 0,Y 354.81,Z 463.501,A -85,B 0,C 180,E1 -13477.892,E2 -13477.892} C_VEL
LIN {X 0,Y 354.916,Z 463.487,A -85,B 0,C 180,E1 -13481.891,E2 -13481.891} C_VEL
LIN {X 0,Y 354.935,Z 463.508,A -85,B 0,C 180,E1 -13485.981,E2 -13485.981} C_VEL
LIN {X 0,Y 354.971,Z 463.517,A -85,B 0,C 180,E1 -13489.736,E2 -13489.736} C_VEL
LIN {X 0,Y 355.121,Z 463.498,A -85,B 0,C 180,E1 -13493.18,E2 -13493.18} C_VEL
LIN {X 0,Y 355.238,Z 463.477,A -85,B 0,C 180,E1 -13497.732,E2 -13497.732} C_VEL
LIN {X 0,Y 355.368,Z 463.461,A -85,B 0,C 180,E1 -13500,E2 -13500} C_VEL
LIN {X 0,Y 355.238,Z 463.467,A -85,B 0,C 180,E1 -13502.267,E2 -13502.267} C_VEL
LIN {X 0,Y 355.12,Z 463.481,A -85,B 0,C 180,E1 -13506.819,E2 -13506.819} C_VEL
LIN {X 0,Y 354.97,Z 463.504,A -85,B 0,C 180,E1 -13510.264,E2 -13510.264} C_VEL
LIN {X 0,Y 354.935,Z 463.521,A -85,B 0,C 180,E1 -13514.019,E2 -13514.019} C_VEL
LIN {X 0,Y 354.915,Z 463.525,A -85,B 0,C 180,E1 -13518.108,E2 -13518.108} C_VEL
LIN {X 0,Y 354.819,Z 463.536,A -85,B 0,C 180,E1 -13522.107,E2 -13522.107} C_VEL
LIN {X 0,Y 354.891,Z 463.477,A -85,B 0,C 180,E1 -13525.828,E2 -13525.828} C_VEL
LIN {X 0,Y 354.847,Z 463.528,A -85,B 0,C 180,E1 -13529.679,E2 -13529.679} C_VEL
LIN {X 0,Y 354.799,Z 463.491,A -85,B 0,C 180,E1 -13533.702,E2 -13533.702} C_VEL
LIN {X 0,Y 354.797,Z 463.53,A -85,B 0,C 180,E1 -13536.459,E2 -13536.459} C_VEL
LIN {X 0,Y 354.818,Z 463.539,A -85,B 0,C 180,E1 -13539.424,E2 -13539.424} C_VEL
LIN {X 0,Y 354.829,Z 463.538,A -85,B 0,C 180,E1 -13542.876,E2 -13542.876} C_VEL
LIN {X 0,Y 354.798,Z 463.541,A -85,B 0,C 180,E1 -13546.11,E2 -13546.11} C_VEL
LIN {X 0,Y 354.819,Z 463.539,A -85,B 0,C 180,E1 -13549.185,E2 -13549.185} C_VEL
LIN {X 0,Y 354.803,Z 463.541,A -85,B 0,C 180,E1 -13552.402,E2 -13552.402} C_VEL
LIN {X 0,Y 354.834,Z 463.707,A -85,B 0,C 180,E1 -13555.463,E2 -13555.463} C_VEL
LIN {X 0,Y 355.119,Z 464.869,A -85,B 0,C 180,E1 -13556.065,E2 -13556.065} C_VEL
LIN {X 0,Y 356.459,Z 467.286,A -85,B 0,C 180,E1 -13556.801,E2 -13556.801} C_VEL
LIN {X 0,Y 358.894,Z 469.166,A -85,B 0,C 180,E1 -13557.999,E2 -13557.999} C_VEL
LIN {X 0,Y 360.238,Z 470.11,A -85,B 0,C 180,E1 -13558.684,E2 -13558.684} C_VEL
LIN {X 0,Y 361.832,Z 472.826,A -85,B 0,C 180,E1 -13559.574,E2 -13559.574} C_VEL
LIN {X 0,Y 364.184,Z 474.841,A -85,B 0,C 180,E1 -13560.836,E2 -13560.836} C_VEL
LIN {X 0,Y 365.949,Z 475.984,A -85,B 0,C 180,E1 -13561.799,E2 -13561.799} C_VEL
LIN {X 0,Y 367.848,Z 478.979,A -85,B 0,C 180,E1 -13562.967,E2 -13562.967} C_VEL
LIN {X 0,Y 370.473,Z 481.115,A -85,B 0,C 180,E1 -13564.519,E2 -13564.519} C_VEL
LIN {X 0,Y 371.966,Z 482.053,A -85,B 0,C 180,E1 -13565.402,E2 -13565.402} C_VEL
LIN {X 0,Y 373.912,Z 485.105,A -85,B 0,C 180,E1 -13566.753,E2 -13566.753} C_VEL
LIN {X 0,Y 376.092,Z 486.986,A -85,B 0,C 180,E1 -13568.238,E2 -13568.238} C_VEL
LIN {X 0,Y 378.312,Z 488.331,A -85,B 0,C 180,E1 -13569.806,E2 -13569.806} C_VEL
LIN {X 0,Y 380.04,Z 491.075,A -85,B 0,C 180,E1 -13571.258,E2 -13571.258} C_VEL
LIN {X 0,Y 382.299,Z 493.078,A -85,B 0,C 180,E1 -13573.17,E2 -13573.17} C_VEL
LIN {X 0,Y 384.917,Z 494.617,A -85,B 0,C 180,E1 -13575.595,E2 -13575.595} C_VEL
LIN {X 0,Y 386.567,Z 497.273,A -85,B 0,C 180,E1 -13577.549,E2 -13577.549} C_VEL
LIN {X 0,Y 388.264,Z 498.967,A -85,B 0,C 180,E1 -13579.816,E2 -13579.816} C_VEL
LIN {X 0,Y 389.919,Z 499.833,A -85,B 0,C 180,E1 -13582.447,E2 -13582.447} C_VEL
LIN {X 0,Y 391.1,Z 500.537,A -85,B 0,C 180,E1 -13585.139,E2 -13585.139} C_VEL
LIN {X 0,Y 391.62,Z 500.762,A -85,B 0,C 180,E1 -13586.914,E2 -13586.914} C_VEL
LIN {X 0,Y 391.907,Z 501.012,A -85,B 0,C 180,E1 -13588.972,E2 -13588.972} C_VEL
LIN {X 0,Y 391.907,Z 501.016,A -85,B 0,C 180,E1 -13591.028,E2 -13591.028} C_VEL
LIN {X 0,Y 391.62,Z 500.762,A -85,B 0,C 180,E1 -13593.086,E2 -13593.086} C_VEL
LIN {X 0,Y 391.016,Z 500.414,A -85,B 0,C 180,E1 -13595.156,E2 -13595.156} C_VEL
LIN {X 0,Y 389.919,Z 499.834,A -85,B 0,C 180,E1 -13597.553,E2 -13597.553} C_VEL
LIN {X 0,Y 388.271,Z 498.925,A -85,B 0,C 180,E1 -13600.184,E2 -13600.184} C_VEL
LIN {X 0,Y 386.564,Z 497.286,A -85,B 0,C 180,E1 -13602.454,E2 -13602.454} C_VEL
LIN {X 0,Y 384.531,Z 494.2,A -85,B 0,C 180,E1 -13604.825,E2 -13604.825} C_VEL
LIN {X 0,Y 381.822,Z 492.749,A -85,B 0,C 180,E1 -13607.235,E2 -13607.235} C_VEL
LIN {X 0,Y 379.617,Z 490.511,A -85,B 0,C 180,E1 -13609.117,E2 -13609.117} C_VEL
LIN {X 0,Y 377.962,Z 487.908,A -85,B 0,C 180,E1 -13610.482,E2 -13610.482} C_VEL
LIN {X 0,Y 374.942,Z 486.208,A -85,B 0,C 180,E1 -13612.524,E2 -13612.524} C_VEL
LIN {X 0,Y 372.825,Z 483.688,A -85,B 0,C 180,E1 -13613.975,E2 -13613.975} C_VEL
LIN {X 0,Y 371.651,Z 481.653,A -85,B 0,C 180,E1 -13614.814,E2 -13614.814} C_VEL
LIN {X 0,Y 368.783,Z 479.891,A -85,B 0,C 180,E1 -13616.488,E2 -13616.488} C_VEL
LIN {X 0,Y 366.809,Z 477.501,A -85,B 0,C 180,E1 -13617.686,E2 -13617.686} C_VEL
LIN {X 0,Y 365.562,Z 475.52,A -85,B 0,C 180,E1 -13618.427,E2 -13618.427} C_VEL
LIN {X 0,Y 362.844,Z 473.872,A -85,B 0,C 180,E1 -13619.861,E2 -13619.861} C_VEL
LIN {X 0,Y 360.894,Z 471.493,A -85,B 0,C 180,E1 -13620.93,E2 -13620.93} C_VEL
LIN {X 0,Y 359.925,Z 469.723,A -85,B 0,C 180,E1 -13621.486,E2 -13621.486} C_VEL
LIN {X 0,Y 356.904,Z 467.762,A -85,B 0,C 180,E1 -13622.965,E2 -13622.965} C_VEL
LIN {X 0,Y 355.415,Z 465.672,A -85,B 0,C 180,E1 -13623.737,E2 -13623.737} C_VEL
LIN {X 0,Y 354.945,Z 464.211,A -85,B 0,C 180,E1 -13624.181,E2 -13624.181} C_VEL
LIN {X 0,Y 354.806,Z 463.602,A -85,B 0,C 180,E1 -13624.713,E2 -13624.713} C_VEL
LIN {X 0,Y 354.802,Z 463.541,A -85,B 0,C 180,E1 -13627.882,E2 -13627.882} C_VEL
LIN {X 0,Y 354.81,Z 463.538,A -85,B 0,C 180,E1 -13631.176,E2 -13631.176} C_VEL
LIN {X 0,Y 354.825,Z 463.536,A -85,B 0,C 180,E1 -13634.517,E2 -13634.517} C_VEL
LIN {X 0,Y 354.831,Z 463.537,A -85,B 0,C 180,E1 -13637.669,E2 -13637.669} C_VEL
LIN {X 0,Y 354.846,Z 463.536,A -85,B 0,C 180,E1 -13640.671,E2 -13640.671} C_VEL
LIN {X 0,Y 354.806,Z 463.503,A -85,B 0,C 180,E1 -13644.534,E2 -13644.534} C_VEL
LIN {X 0,Y 354.116,Z 463.578,A -85,B 0,C 180,E1 -13645.481,E2 -13645.481} C_VEL
LIN {X 0,Y 351.22,Z 463.944,A -85,B 0,C 180,E1 -13647.02,E2 -13647.02} C_VEL
LIN {X 0,Y 348.804,Z 464.271,A -85,B 0,C 180,E1 -13648.266,E2 -13648.266} C_VEL
LIN {X 0,Y 347.809,Z 464.412,A -85,B 0,C 180,E1 -13649.231,E2 -13649.231} C_VEL
LIN {X 0,Y 347.749,Z 464.417,A -85,B 0,C 180,E1 -13649.558,E2 -13649.558} C_VEL
LIN {X 0,Y 347.845,Z 464.35,A -85,B 0,C 180,E1 -13652.744,E2 -13652.744} C_VEL
LIN {X 0,Y 347.778,Z 464.402,A -85,B 0,C 180,E1 -13656.162,E2 -13656.162} C_VEL
LIN {X 0,Y 347.799,Z 464.397,A -85,B 0,C 180,E1 -13659.909,E2 -13659.909} C_VEL
LIN {X 0,Y 347.858,Z 464.403,A -85,B 0,C 180,E1 -13662.359,E2 -13662.359} C_VEL
LIN {X 0,Y 347.89,Z 464.398,A -85,B 0,C 180,E1 -13665.971,E2 -13665.971} C_VEL
LIN {X 0,Y 347.92,Z 464.38,A -85,B 0,C 180,E1 -13669.526,E2 -13669.526} C_VEL
LIN {X 0,Y 348.086,Z 464.359,A -85,B 0,C 180,E1 -13673.042,E2 -13673.042} C_VEL
LIN {X 0,Y 348.201,Z 464.346,A -85,B 0,C 180,E1 -13677.687,E2 -13677.687} C_VEL
LIN {X 0,Y 348.318,Z 464.34,A -85,B 0,C 180,E1 -13680,E2 -13680} C_VEL
LIN {X 0,Y 348.2,Z 464.355,A -85,B 0,C 180,E1 -13682.314,E2 -13682.314} C_VEL
LIN {X 0,Y 348.086,Z 464.372,A -85,B 0,C 180,E1 -13686.958,E2 -13686.958} C_VEL
LIN {X 0,Y 347.921,Z 464.393,A -85,B 0,C 180,E1 -13690.475,E2 -13690.475} C_VEL
LIN {X 0,Y 347.892,Z 464.386,A -85,B 0,C 180,E1 -13694.15,E2 -13694.15} C_VEL
LIN {X 0,Y 347.884,Z 464.356,A -85,B 0,C 180,E1 -13698.291,E2 -13698.291} C_VEL
LIN {X 0,Y 347.761,Z 464.366,A -85,B 0,C 180,E1 -13701.627,E2 -13701.627} C_VEL
LIN {X 0,Y 347.806,Z 464.408,A -85,B 0,C 180,E1 -13705.109,E2 -13705.109} C_VEL
LIN {X 0,Y 347.806,Z 464.358,A -85,B 0,C 180,E1 -13707.694,E2 -13707.694} C_VEL
LIN {X 0,Y 347.765,Z 464.387,A -85,B 0,C 180,E1 -13710.346,E2 -13710.346} C_VEL
LIN {X 0,Y 347.743,Z 464.389,A -85,B 0,C 180,E1 -13714.044,E2 -13714.044} C_VEL
LIN {X 0,Y 347.761,Z 464.417,A -85,B 0,C 180,E1 -13717.321,E2 -13717.321} C_VEL
LIN {X 0,Y 347.789,Z 464.386,A -85,B 0,C 180,E1 -13720.289,E2 -13720.289} C_VEL
LIN {X 0,Y 347.793,Z 464.473,A -85,B 0,C 180,E1 -13723.099,E2 -13723.099} C_VEL
LIN {X 0,Y 349.308,Z 469.322,A -85,B 0,C 180,E1 -13724.764,E2 -13724.764} C_VEL
LIN {X 0,Y 351.622,Z 477.168,A -85,B 0,C 180,E1 -13727.137,E2 -13727.137} C_VEL
LIN {X 0,Y 360.497,Z 492.597,A -85,B 0,C 180,E1 -13728.851,E2 -13728.851} C_VEL
LIN {X 0,Y 369.863,Z 510.427,A -85,B 0,C 180,E1 -13730.538,E2 -13730.538} C_VEL
LIN {X 0,Y 377.248,Z 526.047,A -85,B 0,C 180,E1 -13731.819,E2 -13731.819} C_VEL
LIN {X 0,Y 379.354,Z 535.399,A -85,B 0,C 180,E1 -13732.286,E2 -13732.286} C_VEL
LIN {X 0,Y 374.612,Z 678.072,A -85,B 0,C 180,E1 -13735.056,E2 -13735.056} C_VEL
LIN {X 0,Y 373.542,Z 699.53,A -85,B 0,C 180,E1 -13735.556,E2 -13735.556} C_VEL
LIN {X 0,Y 372.264,Z 713.767,A -85,B 0,C 180,E1 -13736.047,E2 -13736.047} C_VEL
LIN {X 0,Y 370.808,Z 727.171,A -85,B 0,C 180,E1 -13736.658,E2 -13736.658} C_VEL
LIN {X 0,Y 369.215,Z 739.979,A -85,B 0,C 180,E1 -13737.39,E2 -13737.39} C_VEL
LIN {X 0,Y 367.337,Z 752.617,A -85,B 0,C 180,E1 -13738.256,E2 -13738.256} C_VEL
LIN {X 0,Y 365.454,Z 764.259,A -85,B 0,C 180,E1 -13739.202,E2 -13739.202} C_VEL
LIN {X 0,Y 363.159,Z 776.973,A -85,B 0,C 180,E1 -13740.416,E2 -13740.416} C_VEL
LIN {X 0,Y 360.997,Z 788.227,A -85,B 0,C 180,E1 -13741.671,E2 -13741.671} C_VEL
LIN {X 0,Y 358.742,Z 799.067,A -85,B 0,C 180,E1 -13743.062,E2 -13743.062} C_VEL
LIN {X 0,Y 356.579,Z 809.531,A -85,B 0,C 180,E1 -13744.617,E2 -13744.617} C_VEL
LIN {X 0,Y 354.899,Z 817.967,A -85,B 0,C 180,E1 -13746.049,E2 -13746.049} C_VEL
LIN {X 0,Y 352.953,Z 826.925,A -85,B 0,C 180,E1 -13747.77,E2 -13747.77} C_VEL
LIN {X 0,Y 351.348,Z 834.819,A -85,B 0,C 180,E1 -13749.51,E2 -13749.51} C_VEL
LIN {X 0,Y 349.87,Z 842.84,A -85,B 0,C 180,E1 -13751.556,E2 -13751.556} C_VEL
LIN {X 0,Y 348.607,Z 849.744,A -85,B 0,C 180,E1 -13753.606,E2 -13753.606} C_VEL
LIN {X 0,Y 347.824,Z 854.876,A -85,B 0,C 180,E1 -13755.371,E2 -13755.371} C_VEL
LIN {X 0,Y 347.204,Z 859.347,A -85,B 0,C 180,E1 -13757.135,E2 -13757.135} C_VEL
LIN {X 0,Y 346.541,Z 864.242,A -85,B 0,C 180,E1 -13759.483,E2 -13759.483} C_VEL
LIN {X 0,Y 346.282,Z 868.093,A -85,B 0,C 180,E1 -13761.833,E2 -13761.833} C_VEL
LIN {X 0,Y 346.179,Z 870.942,A -85,B 0,C 180,E1 -13764.174,E2 -13764.174} C_VEL
LIN {X 0,Y 346.115,Z 872.822,A -85,B 0,C 180,E1 -13766.508,E2 -13766.508} C_VEL
LIN {X 0,Y 346.07,Z 873.495,A -85,B 0,C 180,E1 -13767.672,E2 -13767.672} C_VEL
LIN {X 0,Y 346.103,Z 873.968,A -85,B 0,C 180,E1 -13770,E2 -13770} C_VEL
LIN {X 0,Y 346.07,Z 873.495,A -85,B 0,C 180,E1 -13772.328,E2 -13772.328} C_VEL
LIN {X 0,Y 346.122,Z 872.075,A -85,B 0,C 180,E1 -13774.659,E2 -13774.659} C_VEL
LIN {X 0,Y 346.216,Z 869.693,A -85,B 0,C 180,E1 -13776.996,E2 -13776.996} C_VEL
LIN {X 0,Y 346.474,Z 865.282,A -85,B 0,C 180,E1 -13779.928,E2 -13779.928} C_VEL
LIN {X 0,Y 346.839,Z 861.918,A -85,B 0,C 180,E1 -13781.691,E2 -13781.691} C_VEL
LIN {X 0,Y 347.576,Z 856.42,A -85,B 0,C 180,E1 -13784.042,E2 -13784.042} C_VEL
LIN {X 0,Y 348.331,Z 851.561,A -85,B 0,C 180,E1 -13785.805,E2 -13785.805} C_VEL
LIN {X 0,Y 349.729,Z 843.895,A -85,B 0,C 180,E1 -13788.148,E2 -13788.148} C_VEL
LIN {X 0,Y 350.914,Z 837.239,A -85,B 0,C 180,E1 -13789.905,E2 -13789.905} C_VEL
LIN {X 0,Y 352.389,Z 829.684,A -85,B 0,C 180,E1 -13791.651,E2 -13791.651} C_VEL
LIN {X 0,Y 354.274,Z 821.101,A -85,B 0,C 180,E1 -13793.375,E2 -13793.375} C_VEL
LIN {X 0,Y 356.259,Z 811.311,A -85,B 0,C 180,E1 -13795.095,E2 -13795.095} C_VEL
LIN {X 0,Y 358.517,Z 800.073,A -85,B 0,C 180,E1 -13796.799,E2 -13796.799} C_VEL
LIN {X 0,Y 360.551,Z 790.515,A -85,B 0,C 180,E1 -13798.05,E2 -13798.05} C_VEL
LIN {X 0,Y 362.555,Z 779.963,A -85,B 0,C 180,E1 -13799.272,E2 -13799.272} C_VEL
LIN {X 0,Y 364.643,Z 768.759,A -85,B 0,C 180,E1 -13800.392,E2 -13800.392} C_VEL
LIN {X 0,Y 366.49,Z 757.842,A -85,B 0,C 180,E1 -13801.342,E2 -13801.342} C_VEL
LIN {X 0,Y 368.578,Z 744.082,A -85,B 0,C 180,E1 -13802.349,E2 -13802.349} C_VEL
LIN {X 0,Y 370.352,Z 730.874,A -85,B 0,C 180,E1 -13803.144,E2 -13803.144} C_VEL
LIN {X 0,Y 371.802,Z 718.283,A -85,B 0,C 180,E1 -13803.76,E2 -13803.76} C_VEL
LIN {X 0,Y 373.079,Z 705.175,A -85,B 0,C 180,E1 -13804.262,E2 -13804.262} C_VEL
LIN {X 0,Y 374.006,Z 692.073,A -85,B 0,C 180,E1 -13804.64,E2 -13804.64} C_VEL
LIN {X 0,Y 375.377,Z 654.788,A -85,B 0,C 180,E1 -13805.395,E2 -13805.395} C_VEL
LIN {X 0,Y 379.354,Z 535.498,A -85,B 0,C 180,E1 -13807.712,E2 -13807.712} C_VEL
LIN {X 0,Y 376.981,Z 525.395,A -85,B 0,C 180,E1 -13808.228,E2 -13808.228} C_VEL
LIN {X 0,Y 368.454,Z 507.66,A -85,B 0,C 180,E1 -13809.71,E2 -13809.71} C_VEL
LIN {X 0,Y 359.626,Z 491.076,A -85,B 0,C 180,E1 -13811.309,E2 -13811.309} C_VEL
LIN {X 0,Y 353.253,Z 480.284,A -85,B 0,C 180,E1 -13812.507,E2 -13812.507} C_VEL
LIN {X 0,Y 351.546,Z 476.973,A -85,B 0,C 180,E1 -13812.899,E2 -13812.899} C_VEL
LIN {X 0,Y 348.938,Z 468.273,A -85,B 0,C 180,E1 -13815.581,E2 -13815.581} C_VEL
LIN {X 0,Y 347.796,Z 464.491,A -85,B 0,C 180,E1 -13816.901,E2 -13816.901} C_VEL
LIN {X 0,Y 347.781,Z 464.387,A -85,B 0,C 180,E1 -13820.165,E2 -13820.165} C_VEL
LIN {X 0,Y 347.784,Z 464.384,A -85,B 0,C 180,E1 -13824.124,E2 -13824.124} C_VEL
LIN {X 0,Y 347.758,Z 464.416,A -85,B 0,C 180,E1 -13828.302,E2 -13828.302} C_VEL
LIN {X 0,Y 347.8,Z 464.359,A -85,B 0,C 180,E1 -13830.99,E2 -13830.99} C_VEL
LIN {X 0,Y 347.825,Z 464.377,A -85,B 0,C 180,E1 -13833.607,E2 -13833.607} C_VEL
LIN {X 0,Y 347.779,Z 464.411,A -85,B 0,C 180,E1 -13836.161,E2 -13836.161} C_VEL
LIN {X 0,Y 347.799,Z 464.345,A -85,B 0,C 180,E1 -13839.908,E2 -13839.908} C_VEL
LIN {X 0,Y 347.859,Z 464.376,A -85,B 0,C 180,E1 -13842.359,E2 -13842.359} C_VEL
LIN {X 0,Y 347.891,Z 464.385,A -85,B 0,C 180,E1 -13845.97,E2 -13845.97} C_VEL
LIN {X 0,Y 347.921,Z 464.394,A -85,B 0,C 180,E1 -13849.525,E2 -13849.525} C_VEL
LIN {X 0,Y 348.086,Z 464.373,A -85,B 0,C 180,E1 -13853.042,E2 -13853.042} C_VEL
LIN {X 0,Y 348.2,Z 464.354,A -85,B 0,C 180,E1 -13857.686,E2 -13857.686} C_VEL
LIN {X 0,Y 348.318,Z 464.338,A -85,B 0,C 180,E1 -13860,E2 -13860} C_VEL
LIN {X 0,Y 348.201,Z 464.344,A -85,B 0,C 180,E1 -13862.313,E2 -13862.313} C_VEL
LIN {X 0,Y 348.086,Z 464.357,A -85,B 0,C 180,E1 -13866.958,E2 -13866.958} C_VEL
LIN {X 0,Y 347.92,Z 464.379,A -85,B 0,C 180,E1 -13870.474,E2 -13870.474} C_VEL
LIN {X 0,Y 347.891,Z 464.399,A -85,B 0,C 180,E1 -13874.15,E2 -13874.15} C_VEL
LIN {X 0,Y 347.883,Z 464.402,A -85,B 0,C 180,E1 -13878.29,E2 -13878.29} C_VEL
LIN {X 0,Y 347.768,Z 464.411,A -85,B 0,C 180,E1 -13881.629,E2 -13881.629} C_VEL
LIN {X 0,Y 347.803,Z 464.369,A -85,B 0,C 180,E1 -13885.109,E2 -13885.109} C_VEL
LIN {X 0,Y 347.805,Z 464.36,A -85,B 0,C 180,E1 -13887.694,E2 -13887.694} C_VEL
LIN {X 0,Y 347.757,Z 464.417,A -85,B 0,C 180,E1 -13890.347,E2 -13890.347} C_VEL
LIN {X 0,Y 347.737,Z 464.37,A -85,B 0,C 180,E1 -13894.464,E2 -13894.464} C_VEL
LIN {X 0,Y 347.775,Z 464.416,A -85,B 0,C 180,E1 -13897.991,E2 -13897.991} C_VEL
LIN {X 0,Y 347.777,Z 464.417,A -85,B 0,C 180,E1 -13901.826,E2 -13901.826} C_VEL
LIN {X 0,Y 347.792,Z 464.414,A -85,B 0,C 180,E1 -13905.012,E2 -13905.012} C_VEL
LIN {X 0,Y 347.762,Z 464.416,A -85,B 0,C 180,E1 -13908.394,E2 -13908.394} C_VEL
LIN {X 0,Y 347.78,Z 464.46,A -85,B 0,C 180,E1 -13912.348,E2 -13912.348} C_VEL
LIN {X 0,Y 347.877,Z 465.191,A -85,B 0,C 180,E1 -13912.948,E2 -13912.948} C_VEL
LIN {X 0,Y 349.47,Z 468.215,A -85,B 0,C 180,E1 -13913.873,E2 -13913.873} C_VEL
LIN {X 0,Y 352.251,Z 470.207,A -85,B 0,C 180,E1 -13915.149,E2 -13915.149} C_VEL
LIN {X 0,Y 353.164,Z 471.125,A -85,B 0,C 180,E1 -13915.597,E2 -13915.597} C_VEL
LIN {X 0,Y 354.797,Z 473.845,A -85,B 0,C 180,E1 -13916.455,E2 -13916.455} C_VEL
LIN {X 0,Y 357.394,Z 475.956,A -85,B 0,C 180,E1 -13917.733,E2 -13917.733} C_VEL
LIN {X 0,Y 358.657,Z 476.773,A -85,B 0,C 180,E1 -13918.343,E2 -13918.343} C_VEL
LIN {X 0,Y 360.381,Z 479.581,A -85,B 0,C 180,E1 -13919.315,E2 -13919.315} C_VEL
LIN {X 0,Y 362.871,Z 481.723,A -85,B 0,C 180,E1 -13920.638,E2 -13920.638} C_VEL
LIN {X 0,Y 364.458,Z 482.665,A -85,B 0,C 180,E1 -13921.479,E2 -13921.479} C_VEL
LIN {X 0,Y 366.593,Z 485.846,A -85,B 0,C 180,E1 -13922.765,E2 -13922.765} C_VEL
LIN {X 0,Y 369.443,Z 488.122,A -85,B 0,C 180,E1 -13924.443,E2 -13924.443} C_VEL
LIN {X 0,Y 370.663,Z 488.923,A -85,B 0,C 180,E1 -13925.158,E2 -13925.158} C_VEL
LIN {X 0,Y 372.695,Z 491.972,A -85,B 0,C 180,E1 -13926.549,E2 -13926.549} C_VEL
LIN {X 0,Y 375.119,Z 494.019,A -85,B 0,C 180,E1 -13928.179,E2 -13928.179} C_VEL
LIN {X 0,Y 377.066,Z 495.077,A -85,B 0,C 180,E1 -13929.521,E2 -13929.521} C_VEL
LIN {X 0,Y 378.926,Z 497.966,A -85,B 0,C 180,E1 -13931.066,E2 -13931.066} C_VEL
LIN {X 0,Y 381.564,Z 500.22,A -85,B 0,C 180,E1 -13933.29,E2 -13933.29} C_VEL
LIN {X 0,Y 383.881,Z 501.551,A -85,B 0,C 180,E1 -13935.429,E2 -13935.429} C_VEL
LIN {X 0,Y 385.521,Z 504.187,A -85,B 0,C 180,E1 -13937.364,E2 -13937.364} C_VEL
LIN {X 0,Y 387.376,Z 506.015,A -85,B 0,C 180,E1 -13939.792,E2 -13939.792} C_VEL
LIN {X 0,Y 388.894,Z 506.805,A -85,B 0,C 180,E1 -13942.136,E2 -13942.136} C_VEL
LIN {X 0,Y 390.146,Z 507.474,A -85,B 0,C 180,E1 -13944.833,E2 -13944.833} C_VEL
LIN {X 0,Y 390.753,Z 507.808,A -85,B 0,C 180,E1 -13946.907,E2 -13946.907} C_VEL
LIN {X 0,Y 391.042,Z 508.058,A -85,B 0,C 180,E1 -13948.97,E2 -13948.97} C_VEL
LIN {X 0,Y 391.042,Z 508.062,A -85,B 0,C 180,E1 -13951.03,E2 -13951.03} C_VEL
LIN {X 0,Y 390.753,Z 507.808,A -85,B 0,C 180,E1 -13953.093,E2 -13953.093} C_VEL
LIN {X 0,Y 390.146,Z 507.466,A -85,B 0,C 180,E1 -13955.167,E2 -13955.167} C_VEL
LIN {X 0,Y 388.894,Z 506.806,A -85,B 0,C 180,E1 -13957.864,E2 -13957.864} C_VEL
LIN {X 0,Y 387.212,Z 505.84,A -85,B 0,C 180,E1 -13960.457,E2 -13960.457} C_VEL
LIN {X 0,Y 385.521,Z 504.196,A -85,B 0,C 180,E1 -13962.636,E2 -13962.636} C_VEL
LIN {X 0,Y 383.616,Z 501.254,A -85,B 0,C 180,E1 -13964.861,E2 -13964.861} C_VEL
LIN {X 0,Y 380.716,Z 499.651,A -85,B 0,C 180,E1 -13967.435,E2 -13967.435} C_VEL
LIN {X 0,Y 378.503,Z 497.423,A -85,B 0,C 180,E1 -13969.282,E2 -13969.282} C_VEL
LIN {X 0,Y 376.661,Z 494.713,A -85,B 0,C 180,E1 -13970.763,E2 -13970.763} C_VEL
LIN {X 0,Y 373.826,Z 493.155,A -85,B 0,C 180,E1 -13972.668,E2 -13972.668} C_VEL
LIN {X 0,Y 371.6,Z 490.602,A -85,B 0,C 180,E1 -13974.176,E2 -13974.176} C_VEL
LIN {X 0,Y 370.471,Z 488.6,A -85,B 0,C 180,E1 -13974.968,E2 -13974.968} C_VEL
LIN {X 0,Y 367.512,Z 486.772,A -85,B 0,C 180,E1 -13976.688,E2 -13976.688} C_VEL
LIN {X 0,Y 365.338,Z 484.197,A -85,B 0,C 180,E1 -13977.982,E2 -13977.982} C_VEL
LIN {X 0,Y 364.229,Z 482.404,A -85,B 0,C 180,E1 -13978.657,E2 -13978.657} C_VEL
LIN {X 0,Y 361.3,Z 480.527,A -85,B 0,C 180,E1 -13980.199,E2 -13980.199} C_VEL
LIN {X 0,Y 359.177,Z 477.877,A -85,B 0,C 180,E1 -13981.341,E2 -13981.341} C_VEL
LIN {X 0,Y 358.303,Z 476.338,A -85,B 0,C 180,E1 -13981.849,E2 -13981.849} C_VEL
LIN {X 0,Y 355.547,Z 474.607,A -85,B 0,C 180,E1 -13983.18,E2 -13983.18} C_VEL
LIN {X 0,Y 353.674,Z 472.193,A -85,B 0,C 180,E1 -13984.117,E2 -13984.117} C_VEL
LIN {X 0,Y 352.639,Z 470.416,A -85,B 0,C 180,E1 -13984.678,E2 -13984.678} C_VEL
LIN {X 0,Y 349.631,Z 468.407,A -85,B 0,C 180,E1 -13986.046,E2 -13986.046} C_VEL
LIN {X 0,Y 348.194,Z 466.134,A -85,B 0,C 180,E1 -13986.759,E2 -13986.759} C_VEL
LIN {X 0,Y 347.845,Z 464.99,A -85,B 0,C 180,E1 -13987.14,E2 -13987.14} C_VEL
LIN {X 0,Y 347.78,Z 464.461,A -85,B 0,C 180,E1 -13987.652,E2 -13987.652} C_VEL
LIN {X 0,Y 347.762,Z 464.416,A -85,B 0,C 180,E1 -13991.606,E2 -13991.606} C_VEL
LIN {X 0,Y 347.793,Z 464.415,A -85,B 0,C 180,E1 -13995.011,E2 -13995.011} C_VEL
LIN {X 0,Y 347.778,Z 464.416,A -85,B 0,C 180,E1 -13998.391,E2 -13998.391} C_VEL
LIN {X 0,Y 347.775,Z 464.416,A -85,B 0,C 180,E1 -14002.009,E2 -14002.009} C_VEL
LIN {X 0,Y 347.737,Z 464.37,A -85,B 0,C 180,E1 -14005.536,E2 -14005.536} C_VEL
LIN {X 0,Y 347.749,Z 464.417,A -85,B 0,C 180,E1 -14009.558,E2 -14009.558} C_VEL
LIN {X 0,Y 347.143,Z 464.497,A -85,B 0,C 180,E1 -14010.526,E2 -14010.526} C_VEL
LIN {X 0,Y 344.318,Z 464.822,A -85,B 0,C 180,E1 -14012.1,E2 -14012.1} C_VEL
LIN {X 0,Y 341.888,Z 465.099,A -85,B 0,C 180,E1 -14013.375,E2 -14013.375} C_VEL
LIN {X 0,Y 340.839,Z 465.227,A -85,B 0,C 180,E1 -14014.362,E2 -14014.362} C_VEL
LIN {X 0,Y 340.752,Z 465.241,A -85,B 0,C 180,E1 -14014.696,E2 -14014.696} C_VEL
LIN {X 0,Y 340.734,Z 465.289,A -85,B 0,C 180,E1 -14018.207,E2 -14018.207} C_VEL
LIN {X 0,Y 340.85,Z 465.276,A -85,B 0,C 180,E1 -14021.984,E2 -14021.984} C_VEL
LIN {X 0,Y 340.862,Z 465.271,A -85,B 0,C 180,E1 -14025.705,E2 -14025.705} C_VEL
LIN {X 0,Y 340.863,Z 465.257,A -85,B 0,C 180,E1 -14029.306,E2 -14029.306} C_VEL
LIN {X 0,Y 341.054,Z 465.236,A -85,B 0,C 180,E1 -14032.898,E2 -14032.898} C_VEL
LIN {X 0,Y 341.163,Z 465.223,A -85,B 0,C 180,E1 -14037.639,E2 -14037.639} C_VEL
LIN {X 0,Y 341.269,Z 465.217,A -85,B 0,C 180,E1 -14040,E2 -14040} C_VEL
LIN {X 0,Y 341.162,Z 465.231,A -85,B 0,C 180,E1 -14042.362,E2 -14042.362} C_VEL
LIN {X 0,Y 341.054,Z 465.244,A -85,B 0,C 180,E1 -14047.102,E2 -14047.102} C_VEL
LIN {X 0,Y 340.864,Z 465.272,A -85,B 0,C 180,E1 -14050.694,E2 -14050.694} C_VEL
LIN {X 0,Y 340.856,Z 465.264,A -85,B 0,C 180,E1 -14054.325,E2 -14054.325} C_VEL
LIN {X 0,Y 340.83,Z 465.229,A -85,B 0,C 180,E1 -14058.467,E2 -14058.467} C_VEL
LIN {X 0,Y 340.711,Z 465.246,A -85,B 0,C 180,E1 -14061.842,E2 -14061.842} C_VEL
LIN {X 0,Y 340.766,Z 465.273,A -85,B 0,C 180,E1 -14065.665,E2 -14065.665} C_VEL
LIN {X 0,Y 340.736,Z 465.234,A -85,B 0,C 180,E1 -14068.32,E2 -14068.32} C_VEL
LIN {X 0,Y 340.71,Z 465.282,A -85,B 0,C 180,E1 -14071.043,E2 -14071.043} C_VEL
LIN {X 0,Y 340.713,Z 465.259,A -85,B 0,C 180,E1 -14075.279,E2 -14075.279} C_VEL
LIN {X 0,Y 340.71,Z 465.284,A -85,B 0,C 180,E1 -14078.388,E2 -14078.388} C_VEL
LIN {X 0,Y 340.722,Z 465.276,A -85,B 0,C 180,E1 -14081.304,E2 -14081.304} C_VEL
LIN {X 0,Y 340.755,Z 465.353,A -85,B 0,C 180,E1 -14082.188,E2 -14082.188} C_VEL
LIN {X 0,Y 343.532,Z 474.492,A -85,B 0,C 180,E1 -14085.31,E2 -14085.31} C_VEL
LIN {X 0,Y 344.331,Z 476.945,A -85,B 0,C 180,E1 -14086.011,E2 -14086.011} C_VEL
LIN {X 0,Y 353.578,Z 492.741,A -85,B 0,C 180,E1 -14087.875,E2 -14087.875} C_VEL
LIN {X 0,Y 362.659,Z 509.677,A -85,B 0,C 180,E1 -14089.582,E2 -14089.582} C_VEL
LIN {X 0,Y 370.781,Z 526.536,A -85,B 0,C 180,E1 -14091.046,E2 -14091.046} C_VEL
LIN {X 0,Y 372.17,Z 529.946,A -85,B 0,C 180,E1 -14091.3,E2 -14091.3} C_VEL
LIN {X 0,Y 373.697,Z 537.264,A -85,B 0,C 180,E1 -14091.661,E2 -14091.661} C_VEL
LIN {X 0,Y 368.739,Z 679.653,A -85,B 0,C 180,E1 -14094.458,E2 -14094.458} C_VEL
LIN {X 0,Y 367.705,Z 699.32,A -85,B 0,C 180,E1 -14094.93,E2 -14094.93} C_VEL
LIN {X 0,Y 366.317,Z 714.124,A -85,B 0,C 180,E1 -14095.45,E2 -14095.45} C_VEL
LIN {X 0,Y 364.87,Z 726.96,A -85,B 0,C 180,E1 -14096.043,E2 -14096.043} C_VEL
LIN {X 0,Y 363.2,Z 739.768,A -85,B 0,C 180,E1 -14096.781,E2 -14096.781} C_VEL
LIN {X 0,Y 361.273,Z 752.405,A -85,B 0,C 180,E1 -14097.659,E2 -14097.659} C_VEL
LIN {X 0,Y 359.337,Z 764.048,A -85,B 0,C 180,E1 -14098.619,E2 -14098.619} C_VEL
LIN {X 0,Y 356.909,Z 776.883,A -85,B 0,C 180,E1 -14099.861,E2 -14099.861} C_VEL
LIN {X 0,Y 354.672,Z 788.014,A -85,B 0,C 180,E1 -14101.119,E2 -14101.119} C_VEL
LIN {X 0,Y 352.359,Z 798.855,A -85,B 0,C 180,E1 -14102.534,E2 -14102.534} C_VEL
LIN {X 0,Y 350.077,Z 809.316,A -85,B 0,C 180,E1 -14104.111,E2 -14104.111} C_VEL
LIN {X 0,Y 348.261,Z 817.971,A -85,B 0,C 180,E1 -14105.607,E2 -14105.607} C_VEL
LIN {X 0,Y 346.277,Z 826.712,A -85,B 0,C 180,E1 -14107.318,E2 -14107.318} C_VEL
LIN {X 0,Y 344.596,Z 834.606,A -85,B 0,C 180,E1 -14109.09,E2 -14109.09} C_VEL
LIN {X 0,Y 343.191,Z 841.572,A -85,B 0,C 180,E1 -14110.874,E2 -14110.874} C_VEL
LIN {X 0,Y 342.049,Z 847.715,A -85,B 0,C 180,E1 -14112.667,E2 -14112.667} C_VEL
LIN {X 0,Y 340.865,Z 854.663,A -85,B 0,C 180,E1 -14115.065,E2 -14115.065} C_VEL
LIN {X 0,Y 339.984,Z 860.42,A -85,B 0,C 180,E1 -14117.464,E2 -14117.464} C_VEL
LIN {X 0,Y 339.489,Z 864.03,A -85,B 0,C 180,E1 -14119.262,E2 -14119.262} C_VEL
LIN {X 0,Y 339.208,Z 867.882,A -85,B 0,C 180,E1 -14121.661,E2 -14121.661} C_VEL
LIN {X 0,Y 339.076,Z 870.876,A -85,B 0,C 180,E1 -14124.204,E2 -14124.204} C_VEL
LIN {X 0,Y 339.039,Z 872.612,A -85,B 0,C 180,E1 -14126.435,E2 -14126.435} C_VEL
LIN {X 0,Y 338.985,Z 873.286,A -85,B 0,C 180,E1 -14127.624,E2 -14127.624} C_VEL
LIN {X 0,Y 339.006,Z 873.758,A -85,B 0,C 180,E1 -14130,E2 -14130} C_VEL
LIN {X 0,Y 338.985,Z 873.286,A -85,B 0,C 180,E1 -14132.376,E2 -14132.376} C_VEL
LIN {X 0,Y 339.027,Z 871.865,A -85,B 0,C 180,E1 -14134.756,E2 -14134.756} C_VEL
LIN {X 0,Y 339.13,Z 869.482,A -85,B 0,C 180,E1 -14137.143,E2 -14137.143} C_VEL
LIN {X 0,Y 339.402,Z 865.07,A -85,B 0,C 180,E1 -14140.137,E2 -14140.137} C_VEL
LIN {X 0,Y 339.817,Z 861.706,A -85,B 0,C 180,E1 -14141.936,E2 -14141.936} C_VEL
LIN {X 0,Y 340.596,Z 856.207,A -85,B 0,C 180,E1 -14144.336,E2 -14144.336} C_VEL
LIN {X 0,Y 341.378,Z 851.348,A -85,B 0,C 180,E1 -14146.136,E2 -14146.136} C_VEL
LIN {X 0,Y 342.851,Z 843.681,A -85,B 0,C 180,E1 -14148.525,E2 -14148.525} C_VEL
LIN {X 0,Y 344.102,Z 837.025,A -85,B 0,C 180,E1 -14150.316,E2 -14150.316} C_VEL
LIN {X 0,Y 345.697,Z 829.471,A -85,B 0,C 180,E1 -14152.092,E2 -14152.092} C_VEL
LIN {X 0,Y 347.68,Z 820.889,A -85,B 0,C 180,E1 -14153.845,E2 -14153.845} C_VEL
LIN {X 0,Y 349.719,Z 811.097,A -85,B 0,C 180,E1 -14155.597,E2 -14155.597} C_VEL
LIN {X 0,Y 352.112,Z 799.861,A -85,B 0,C 180,E1 -14157.326,E2 -14157.326} C_VEL
LIN {X 0,Y 354.2,Z 790.306,A -85,B 0,C 180,E1 -14158.598,E2 -14158.598} C_VEL
LIN {X 0,Y 356.537,Z 778.772,A -85,B 0,C 180,E1 -14159.938,E2 -14159.938} C_VEL
LIN {X 0,Y 358.458,Z 768.547,A -85,B 0,C 180,E1 -14160.974,E2 -14160.974} C_VEL
LIN {X 0,Y 360.663,Z 755.888,A -85,B 0,C 180,E1 -14162.072,E2 -14162.072} C_VEL
LIN {X 0,Y 362.589,Z 743.871,A -85,B 0,C 180,E1 -14162.951,E2 -14162.951} C_VEL
LIN {X 0,Y 364.414,Z 730.664,A -85,B 0,C 180,E1 -14163.756,E2 -14163.756} C_VEL
LIN {X 0,Y 365.971,Z 717.581,A -85,B 0,C 180,E1 -14164.4,E2 -14164.4} C_VEL
LIN {X 0,Y 367.229,Z 705.153,A -85,B 0,C 180,E1 -14164.878,E2 -14164.878} C_VEL
LIN {X 0,Y 368.178,Z 691.863,A -85,B 0,C 180,E1 -14165.269,E2 -14165.269} C_VEL
LIN {X 0,Y 369.602,Z 654.578,A -85,B 0,C 180,E1 -14166.034,E2 -14166.034} C_VEL
LIN {X 0,Y 373.66,Z 538.172,A -85,B 0,C 180,E1 -14168.321,E2 -14168.321} C_VEL
LIN {X 0,Y 373.329,Z 535.126,A -85,B 0,C 180,E1 -14168.434,E2 -14168.434} C_VEL
LIN {X 0,Y 371.683,Z 528.465,A -85,B 0,C 180,E1 -14168.795,E2 -14168.795} C_VEL
LIN {X 0,Y 363.27,Z 510.927,A -85,B 0,C 180,E1 -14170.305,E2 -14170.305} C_VEL
LIN {X 0,Y 354.84,Z 495.062,A -85,B 0,C 180,E1 -14171.881,E2 -14171.881} C_VEL
LIN {X 0,Y 348.704,Z 484.545,A -85,B 0,C 180,E1 -14173.073,E2 -14173.073} C_VEL
LIN {X 0,Y 344.263,Z 476.668,A -85,B 0,C 180,E1 -14174.03,E2 -14174.03} C_VEL
LIN {X 0,Y 341.811,Z 468.848,A -85,B 0,C 180,E1 -14176.55,E2 -14176.55} C_VEL
LIN {X 0,Y 340.755,Z 465.38,A -85,B 0,C 180,E1 -14177.812,E2 -14177.812} C_VEL
LIN {X 0,Y 340.729,Z 465.265,A -85,B 0,C 180,E1 -14180.252,E2 -14180.252} C_VEL
LIN {X 0,Y 340.707,Z 465.274,A -85,B 0,C 180,E1 -14183.558,E2 -14183.558} C_VEL
LIN {X 0,Y 340.69,Z 465.269,A -85,B 0,C 180,E1 -14186.153,E2 -14186.153} C_VEL
LIN {X 0,Y 340.77,Z 465.241,A -85,B 0,C 180,E1 -14190.332,E2 -14190.332} C_VEL
